	(*Valve 12, A+B*)
	(*spare*)
		Valve12FB
			(
			Enable_Motion:= Enable_Motion ,
			Enable_Latch:= TRUE,					(*Enabling Runs Valve as detent type (maintained solenoids*)
			Enable_SideA_PreCharge:= FALSE,		(*Enabling Turns Side A PreCharge Active, reset when Side B is energized in Auto*)
			Enable_SideB_PreCharge:= FALSE,		(*Enabling Turns Side B PreCharge Active, reset when Side A is energized in Auto*)
			PreCharge_Time:= T#0.10S,
			Enable_Auto_Commands:= Enable_Motion,
			Enable_Manual_Commands:= FALSE,
			In_Manual_SideA_Command:= FALSE,
			In_Manual_SideB_Command:= FALSE,
			SideA_Indicator:= FALSE,
			SideB_Indicator:= FALSE,
			TurnOn_SideA_SOL=> N100.Q.22,
			TurnOn_SideB_SOL=> N100.Q.23,
			TurnOn_SideA_Indicator=> ,
			TurnOn_SideB_Indicator=>
			 );
		Valve12FB.In_Auto_SideA_Command:= FALSE;
		Valve12FB.In_Auto_SideB_Command:= FALSE;


	(*Valve 13, A+B*)
	(*spare*)
		Valve13FB
			(
			Enable_Motion:= Enable_Motion ,
			Enable_Latch:= TRUE,					(*Enabling Runs Valve as detent type (maintained solenoids*)
			Enable_SideA_PreCharge:= FALSE,		(*Enabling Turns Side A PreCharge Active, reset when Side B is energized in Auto*)
			Enable_SideB_PreCharge:= FALSE,		(*Enabling Turns Side B PreCharge Active, reset when Side A is energized in Auto*)
			PreCharge_Time:= T#0.10S,
			Enable_Auto_Commands:= Enable_Motion,
			Enable_Manual_Commands:= FALSE,
			In_Manual_SideA_Command:= FALSE,
			In_Manual_SideB_Command:= FALSE,
			SideA_Indicator:= FALSE,
			SideB_Indicator:= FALSE,
			TurnOn_SideA_SOL=> N100.Q.24,
			TurnOn_SideB_SOL=> N100.Q.25,
			TurnOn_SideA_Indicator=> ,
			TurnOn_SideB_Indicator=>
			 );
		Valve13FB.In_Auto_SideA_Command:= FALSE;
		Valve13FB.In_Auto_SideB_Command:= FALSE;


	(*Valve 14, A+B*)
	(*spare*)
		Valve14FB
			(
			Enable_Motion:= Enable_Motion ,
			Enable_Latch:= TRUE,					(*Enabling Runs Valve as detent type (maintained solenoids*)
			Enable_SideA_PreCharge:= FALSE,		(*Enabling Turns Side A PreCharge Active, reset when Side B is energized in Auto*)
			Enable_SideB_PreCharge:= FALSE,		(*Enabling Turns Side B PreCharge Active, reset when Side A is energized in Auto*)
			PreCharge_Time:= T#0.10S,
			Enable_Auto_Commands:= Enable_Motion,
			Enable_Manual_Commands:= FALSE,
			In_Manual_SideA_Command:= FALSE,
			In_Manual_SideB_Command:= FALSE,
			SideA_Indicator:= FALSE,
			SideB_Indicator:= FALSE,
			TurnOn_SideA_SOL=> N100.Q.26,
			TurnOn_SideB_SOL=> N100.Q.27,
			TurnOn_SideA_Indicator=> ,
			TurnOn_SideB_Indicator=>
			 );
		Valve14FB.In_Auto_SideA_Command:= FALSE;
		Valve14FB.In_Auto_SideB_Command:= FALSE;


	(*Valve 15, A+B*)
	(*spare*)
		Valve15FB
			(
			Enable_Motion:= Enable_Motion ,
			Enable_Latch:= TRUE,					(*Enabling Runs Valve as detent type (maintained solenoids*)
			Enable_SideA_PreCharge:= FALSE,		(*Enabling Turns Side A PreCharge Active, reset when Side B is energized in Auto*)
			Enable_SideB_PreCharge:= FALSE,		(*Enabling Turns Side B PreCharge Active, reset when Side A is energized in Auto*)
			PreCharge_Time:= T#0.10S,
			Enable_Auto_Commands:= Enable_Motion,
			Enable_Manual_Commands:= FALSE,
			In_Manual_SideA_Command:= FALSE,
			In_Manual_SideB_Command:= FALSE,
			SideA_Indicator:= FALSE,
			SideB_Indicator:= FALSE,
			TurnOn_SideA_SOL=> N100.Q.28,
			TurnOn_SideB_SOL=> N100.Q.29,
			TurnOn_SideA_Indicator=> ,
			TurnOn_SideB_Indicator=>
			 );
		Valve15FB.In_Auto_SideA_Command:= FALSE;
		Valve15FB.In_Auto_SideB_Command:= FALSE;


	(*Valve 16, A+B*)
	(*spare*)
		Valve16FB
			(
			Enable_Motion:= Enable_Motion ,
			Enable_Latch:= TRUE,					(*Enabling Runs Valve as detent type (maintained solenoids*)
			Enable_SideA_PreCharge:= FALSE,		(*Enabling Turns Side A PreCharge Active, reset when Side B is energized in Auto*)
			Enable_SideB_PreCharge:= FALSE,		(*Enabling Turns Side B PreCharge Active, reset when Side A is energized in Auto*)
			PreCharge_Time:= T#0.10S,
			Enable_Auto_Commands:= Enable_Motion,
			Enable_Manual_Commands:= FALSE,
			In_Manual_SideA_Command:= FALSE,
			In_Manual_SideB_Command:= FALSE,
			SideA_Indicator:= FALSE,
			SideB_Indicator:= FALSE,
			TurnOn_SideA_SOL=> N100.Q.30,
			TurnOn_SideB_SOL=> N100.Q.31,
			TurnOn_SideA_Indicator=> ,
			TurnOn_SideB_Indicator=>
			 );
		Valve16FB.In_Auto_SideA_Command:= FALSE;
		Valve16FB.In_Auto_SideB_Command:= FALSE;


























(*end*)
END_ACTION

ACTION Xfer_To_UI:
	(*Transfer General Status and I/O Images for Display On HMI*)
	Discrete_Image.CLFaults1:= CLFaults1;
	Discrete_Image.CLFaults2:= CLFaults2;
	Discrete_Image.CLFaults3:= CLFaults3;
	Discrete_Image.CLFaults4:= CLFaults4;
	Discrete_Image.CLFaulted:= CLFaulted;
	Discrete_Image.PPFaults:= PPFaults;
	Discrete_Image.PPFaulted:= PPFaulted;

	Discrete_Image.N01:=N01;
	Discrete_Image.N02:=N02;
	Discrete_Image.N03:=N03;
	Discrete_Image.N04:=N04;
	Discrete_Image.N05:=N05;
	Discrete_Image.N06:=N06;
	Discrete_Image.N07:=N07;
	Discrete_Image.N08:=N08;
	Discrete_Image.N09:=N09;
	Discrete_Image.N100:=N100;
	Discrete_Image.N100_STAT:=N100_STAT;
	Discrete_Image.NodeLayout:=NodeLayout;
	Discrete_Image.NodeState:=NodeState;

	Discrete_Image.ID:= ID;
	Discrete_Image.ECatSlave_Cable_Breaks:= ECatSlave_Cable_Breaks;
	Discrete_Image.Input_Node_Count:= Input_Node_Count;
	Discrete_Image.VB_Node_Count:= VB_Node_Count;
















(*end*)
END_ACTION

END_PROGRAM

// ---- POUs/Fixtures and EOAT/Not_Used/EOAT10.TcPOU
(*EOAT*)


PROGRAM EOAT10

VAR_INPUT
(*General Inputs*)
	Enable_FB: BOOL;
	Enable_Motion: BOOL;
	Dry_Cycle: BOOL;
	NodeLayout:udt_ECATNodeData_20221507;
	ID: UINT;

	Input_Node_Count: UDINT;
	Output_Node_Count: UDINT;
	VB_Node_Count: UDINT;
	Robot_WorkingOK: BOOL;

(*CMDs (commands)*)
	CMD_CheckAllSensors_OFF: BOOL;
	CMD_CheckSensorsOFF_Grp1: BOOL;
	CMD_CheckSensorsOFF_Grp2: BOOL;
	CMD_CheckSensorsOFF_Grp3: BOOL;
	CMD_CheckSensorsOFF_Grp4: BOOL;
	CMD_CheckSensorsOFF_Grp5: BOOL;

	CMD_CheckAllSensors_ON: BOOL;
	CMD_CheckSensorsON_Grp1: BOOL;
	CMD_CheckSensorsON_Grp2: BOOL;
	CMD_CheckSensorsON_Grp3: BOOL;
	CMD_CheckSensorsON_Grp4: BOOL;
	CMD_CheckSensorsON_Grp5: BOOL;

	CMD_Tool_To_WORK: BOOL;
	CMD_CylToWORK_Grp1: BOOL;
	CMD_CylToWORK_Grp2: BOOL;
	CMD_CylToWORK_Grp3: BOOL;
	CMD_CylToWORK_Grp4: BOOL;
	CMD_CylToWORK_Grp5: BOOL;

	CMD_Tool_To_HOME: BOOL;
	CMD_CylToHOME_Grp1: BOOL;
	CMD_CylToHOME_Grp2: BOOL;
	CMD_CylToHOME_Grp3: BOOL;
	CMD_CylToHOME_Grp4: BOOL;
	CMD_CylToHOME_Grp5: BOOL;


END_VAR

VAR
(*Hardware Related Data Types*)
			(*Develop "Beckhoff Nodes"*)
			{attribute 'OPC.UA.DA':='1'}
			N01 AT %I*: udt_EP1008_002_v2;
			{attribute 'OPC.UA.DA':='1'}
			N02 AT %I*: udt_EP1008_002_v2;
			{attribute 'OPC.UA.DA':='1'}
			N03 AT %I*: udt_EP1008_002_v2;
			{attribute 'OPC.UA.DA':='1'}
			N04 AT %I*: udt_EP1008_002_v2;
			{attribute 'OPC.UA.DA':='1'}
			N05 AT %I*: udt_EP1008_002_v2;
			{attribute 'OPC.UA.DA':='1'}
			N06 AT %I*: udt_EP1008_002_v2;
			{attribute 'OPC.UA.DA':='1'}
			N07 AT %I*: udt_EP1008_002_v2;
			{attribute 'OPC.UA.DA':='1'}
			N08 AT %I*: udt_EP1008_002_v2;
			{attribute 'OPC.UA.DA':='1'}
			N09 AT %I*: udt_EP1008_002_v2;
			{attribute 'OPC.UA.DA':='1'}
			N100 AT %Q*: udt_SMC_EX260_ValveBank;
			{attribute 'OPC.UA.DA':='1'}
			N100_STAT AT %I*:udt_SMC_EX260_Stat;

(* Nodes States*)
	NodeState: ARRAY[0..63] OF UINT;
	DiscreteNode_OK: BOOL;
(* Cable Break States*)
	ECatSlave_Cable_Breaks: ARRAY[0..1]OF DINT;

(*Standard Internal Variables*)
		(*Generic Sensor Variables*)
		All_Sensors_On: UINT;
		All_Sensors_Off: UINT;
		(*Generic Position Variables*)
		Tool_At_Home: UINT;
		Tool_At_Work: UINT;
		(*General Internals*)
		CLFaulted: UDINT;
		PPFaulted: UDINT;

(*Non-Standard Variables*)

		(*FB Instances*)
		Clamp1FB: FB_Cylinder_Status;
		Clamp2FB: FB_Cylinder_Status;
		Clamp3FB: FB_Cylinder_Status;
		Clamp4FB: FB_Cylinder_Status;
		Clamp5FB: FB_Cylinder_Status;
		Clamp6FB: FB_Cylinder_Status;
		Clamp7FB: FB_Cylinder_Status;
		Clamp8FB: FB_Cylinder_Status;
		Clamp9FB: FB_Cylinder_Status;
		Clamp10FB: FB_Cylinder_Status;
		Clamp11FB: FB_Cylinder_Status;
		Clamp12FB: FB_Cylinder_Status;
		Pin1FB: FB_Cylinder_Status;
		Pin2FB: FB_Cylinder_Status;
		Pin3FB: FB_Cylinder_Status;
		Pin4FB: FB_Cylinder_Status;
		Pin5FB: FB_Cylinder_Status;
		Pin6FB: FB_Cylinder_Status;

		Part_Present1FB: FB_PP_Sensor;
		Part_Present2FB: FB_PP_Sensor;
		Part_Present3FB: FB_PP_Sensor;
		Part_Present4FB: FB_PP_Sensor;
		Part_Present5FB: FB_PP_Sensor;
		Part_Present6FB: FB_PP_Sensor;
		Part_Present7FB: FB_PP_Sensor;
		Part_Present8FB: FB_PP_Sensor;

		(*Valve FBs*)
		Valve1FB: FB_GTAC_Valve_20170704;
		Valve2FB: FB_GTAC_Valve_20170704;
		Valve3FB: FB_GTAC_Valve_20170704;
		Valve4FB: FB_GTAC_Valve_20170704;
		Valve5FB: FB_GTAC_Valve_20170704;
		Valve6FB: FB_GTAC_Valve_20170704;
		Valve7FB: FB_GTAC_Valve_20170704;
		Valve8FB: FB_GTAC_Valve_20170704;
		Valve9FB: FB_GTAC_Valve_20170704;
		Valve10FB: FB_GTAC_Valve_20170704;
		Valve11FB: FB_GTAC_Valve_20170704;
		Valve12FB: FB_GTAC_Valve_20170704;
		Valve13FB: FB_GTAC_Valve_20170704;
		Valve14FB: FB_GTAC_Valve_20170704;
		Valve15FB: FB_GTAC_Valve_20170704;
		Valve16FB: FB_GTAC_Valve_20170704;

		(*Tool Positions*)
		Clamp1ADVD: BOOL;
		Clamp1RETD: BOOL;
		Clamp2ADVD: BOOL;
		Clamp2RETD: BOOL;
		Clamp3ADVD: BOOL;
		Clamp3RETD: BOOL;
		Clamp4ADVD: BOOL;
		Clamp4RETD: BOOL;
		Clamp5ADVD: BOOL;
		Clamp5RETD: BOOL;
		Clamp6ADVD: BOOL;
		Clamp6RETD: BOOL;
		Clamp7ADVD: BOOL;
		Clamp7RETD: BOOL;
		Clamp8ADVD: BOOL;
		Clamp8RETD: BOOL;
		Clamp9ADVD: BOOL;
		Clamp9RETD: BOOL;
		Clamp10ADVD: BOOL;
		Clamp10RETD: BOOL;
		Clamp11ADVD: BOOL;
		Clamp11RETD: BOOL;
		Clamp12ADVD: BOOL;
		Clamp12RETD: BOOL;
		Pin1ADVD: BOOL;
		Pin1RETD: BOOL;
		Pin2ADVD: BOOL;
		Pin2RETD: BOOL;
		Pin3ADVD: BOOL;
		Pin3RETD: BOOL;
		Pin4ADVD: BOOL;
		Pin4RETD: BOOL;
		Pin5ADVD: BOOL;
		Pin5RETD: BOOL;
		Pin6ADVD: BOOL;
		Pin6RETD: BOOL;

		(*Part Present Sensors*)
		(*Main Body Present*)
		Part_Present1: BOOL;
		Part_Present2: BOOL;
		Part_Present3: BOOL;
		Part_Present4: BOOL;
		Part_Present5: BOOL;
		Part_Present6: BOOL;
		Part_Present7: BOOL;
		Part_Present8: BOOL;



END_VAR

VAR_OUTPUT

		FB_OK: BOOL;
		Discrete_Image: udt_EOATxx_Image_20170607;

		EOAT_FLT: BOOL;

		CLFaults1:UDINT;
		CLFaults2:UDINT;
		CLFaults3:UDINT;
		CLFaults4:UDINT;
		PPFaults: UDINT;

		EOAT_All_Empty: BOOL;
		EOAT_Part1_Empty: BOOL;
		EOAT_Part2_Empty: BOOL;
		EOAT_Part3_Empty: BOOL;
		EOAT_Part4_Empty: BOOL;
		EOAT_Part5_Empty: BOOL;

		EOAT_Full: BOOL;
		Part1_In_EOAT: BOOL;
		Part2_In_EOAT: BOOL;
		Part3_In_EOAT: BOOL;
		Part4_In_EOAT: BOOL;
		Part5_In_EOAT: BOOL;

	(*ACKS*)
		ACK_Tool_At_WORK: BOOL;
		ACK_CylAtWORK_Grp1: BOOL;
		ACK_CylAtWORK_Grp2: BOOL;
		ACK_CylAtWORK_Grp3: BOOL;
		ACK_CylAtWORK_Grp4: BOOL;
		ACK_CylAtWORK_Grp5: BOOL;
	
		ACK_Tool_At_HOME: BOOL;
		ACK_CylAtHOME_Grp1: BOOL;
		ACK_CylAtHOME_Grp2: BOOL;
		ACK_CylAtHOME_Grp3: BOOL;
		ACK_CylAtHOME_Grp4: BOOL;
		ACK_CylAtHOME_Grp5: BOOL;


END_VAR

	(*Set FB_OK to True*)
	FB_OK:= TRUE;


(*---------------------------------------------------- Gather Hardwear ------------------------------------------------------*)
	Hardware();


(*---------------------------------------------------- Gather Clamp Sensor Inputs --------------------------------------*)
	Cylinders();


(*---------------------------------------------------- Gather Part Present Sensor Inputs ------------------------------*)
	Proxies();


(*---------------------------------------------------- Group Clamp Sensors -----------------------------------------------*)
	Tool_States();


(*---------------------------------------------------- Group Part Present Sensors ---------------------------------------*)
	All_Sensors();



(*---------------------------------------------------- Status and Faults--------------------------------------------------------*)
	Status_and_Faults();


(*---------------------------------------------------- Transfer to UI -------------------------------------------------------------*)
	Xfer_To_UI();


(*------------------------------------------------------Transfer Valve Outputs ----------------------------------------------*)
	ValveBank1();


(*---------------------------------------------------- Gather Robot Registration-------------------------------------------*)









(*end*)

ACTION All_Sensors:


(*	Note - In the event there is a left part and a right part, grouping the sensors allows only portions of the sensors to be monitored at a time.
		If this is not advantageous to the design, there is still the option to group all the sensors as one group instead.
		In this example, there are all 5 groups set up. 
		Change this section to suit the specific design you have, where .0 is all, .1 is group one, .2 is group two, etc*)


	(*All Sensors Off*)
	All_Sensors_Off.0:= NOT Part_Present1 AND NOT Part_Present2 AND NOT  Part_Present3
					AND NOT Part_Present4 AND NOT Part_Present5 AND NOT Part_Present6
					AND NOT Part_Present7 AND NOT Part_Present8;

	(*All Sensors Off - Group 1*)
	All_Sensors_Off.1:= NOT Part_Present1 AND NOT Part_Present2 AND NOT  Part_Present3
					AND NOT Part_Present4 AND NOT Part_Present5;

	(*All Sensors Off - Group 2*)
	All_Sensors_Off.2:= NOT Part_Present6 AND NOT Part_Present7 AND NOT Part_Present8;

	(*All Sensors Off - Group 3*)
	All_Sensors_Off.3:= FALSE;

	(*All Sensors Off - Group 4*)
	All_Sensors_Off.4:= FALSE;

	(*All Sensors Off - Group 5*)
	All_Sensors_Off.5:= FALSE;



	(*All Sensors On*)
	All_Sensors_On.0:= (Part_Present1 AND Part_Present2 AND Part_Present3
					AND Part_Present4 AND Part_Present5 AND Part_Present6
					AND Part_Present7 AND Part_Present8)
					OR (All_Sensors_Off.0 AND Dry_Cycle);

	(*All Sensors On - Group 1*)
	All_Sensors_On.1:= (Part_Present1 AND Part_Present2 AND Part_Present3 AND Part_Present4 AND Part_Present5)
					OR (All_Sensors_Off.0 AND Dry_Cycle);

	(*All Sensors On - Group 2*)
	All_Sensors_On.2:= (Part_Present6 AND Part_Present7 AND Part_Present8)
					OR (All_Sensors_Off.0 AND Dry_Cycle);

	(*All Sensors On - Group 3*)
	All_Sensors_On.3:= (FALSE)
					OR (All_Sensors_Off.0 AND Dry_Cycle);

	(*All Sensors On - Group 4*)
	All_Sensors_On.4:= (FALSE)
					OR (All_Sensors_Off.0 AND Dry_Cycle);

	(*All Sensors On - Group 5*)
	All_Sensors_On.5:= (FALSE)
					OR (All_Sensors_Off.0 AND Dry_Cycle);




	(*Group all Sensors*)
	IF CMD_CheckAllSensors_OFF AND All_Sensors_Off.0
		THEN
			EOAT_All_Empty:= TRUE;
			EOAT_Full:= FALSE;

	ELSIF CMD_CheckAllSensors_ON AND All_Sensors_On.0
		THEN
			EOAT_All_Empty:= FALSE;
			EOAT_Full:= TRUE;

	END_IF

	IF CMD_CheckSensorsOFF_Grp1 AND All_Sensors_Off.1
		THEN
			EOAT_Part1_Empty:= TRUE;
			Part1_In_EOAT:= FALSE;

	ELSIF CMD_CheckSensorsON_Grp1 AND All_Sensors_On.1
		THEN
			EOAT_Part1_Empty:= FALSE;
			Part1_In_EOAT:= TRUE;

	END_IF

	IF CMD_CheckSensorsOFF_Grp2 AND All_Sensors_Off.2
		THEN
			EOAT_Part2_Empty:= TRUE;
			Part2_In_EOAT:= FALSE;

	ELSIF CMD_CheckSensorsON_Grp2 AND All_Sensors_On.2
		THEN
			EOAT_Part2_Empty:= FALSE;
			Part2_In_EOAT:= TRUE;

	END_IF

	IF CMD_CheckSensorsOFF_Grp3 AND All_Sensors_Off.3
		THEN
			EOAT_Part3_Empty:= TRUE;
			Part3_In_EOAT:= FALSE;

	ELSIF CMD_CheckSensorsON_Grp3 AND All_Sensors_On.3
		THEN
			EOAT_Part3_Empty:= FALSE;
			Part3_In_EOAT:= TRUE;

	ELSIF CMD_CheckSensorsON_Grp3 AND All_Sensors_On.3
		THEN
			EOAT_Part3_Empty:= FALSE;
			Part3_In_EOAT:= TRUE;

	END_IF

	IF CMD_CheckSensorsOFF_Grp4 AND All_Sensors_Off.4
		THEN
			EOAT_Part4_Empty:= TRUE;
			Part4_In_EOAT:= FALSE;
	ELSIF CMD_CheckSensorsON_Grp4 AND All_Sensors_On.4
		THEN
			EOAT_Part4_Empty:= FALSE;
			Part4_In_EOAT:= TRUE;

	END_IF

	IF CMD_CheckSensorsOFF_Grp5 AND All_Sensors_Off.5
		THEN
			EOAT_Part5_Empty:= TRUE;
			Part5_In_EOAT:= FALSE;
	ELSIF CMD_CheckSensorsON_Grp5 AND All_Sensors_On.5
		THEN
			EOAT_Part5_Empty:= FALSE;
			Part5_In_EOAT:= TRUE;

	END_IF












(*end*)
END_ACTION

ACTION Cylinders:
(*Clamps*)(*Clamps*)(*Clamps*)
(*Clamps*)(*Clamps*)(*Clamps*)
(*Clamps*)(*Clamps*)(*Clamps*)

		(*Clamp1*)
		Clamp1FB(
			Retracted_Sensor:= N02.I.0,
			Advanced_Sensor:= N02.I.1,
			Retract_Solenoid:= N100.Q.1,
			Advance_Solenoid:= N100.Q.0,
			Ret_Delay:= T#0.1s,
			Adv_Delay:= T#0.1s,
			Fault_Delay:= T#3s,
			Disable_Fault:= FALSE,
			In_Retracted_Position=> Clamp1RETD,
			In_Advanced_Position=> Clamp1ADVD,
			Faulted=> CLFaults1.1 );

		(*Clamp2 *)
		Clamp2FB(
			Retracted_Sensor:= N02.I.2,
			Advanced_Sensor:= N02.I.3,
			Retract_Solenoid:= N100.Q.1,
			Advance_Solenoid:= N100.Q.0,
			Ret_Delay:= T#0.1s,
			Adv_Delay:= T#0.1s,
			Fault_Delay:= T#3s,
			Disable_Fault:= FALSE,
			In_Retracted_Position=> Clamp2RETD,
			In_Advanced_Position=> Clamp2ADVD,
			Faulted=> CLFaults1.2 );

		(*Clamp3 *)
		Clamp3FB(
			Retracted_Sensor:= N02.I.4,
			Advanced_Sensor:= N02.I.5,
			Retract_Solenoid:= N100.Q.5,
			Advance_Solenoid:= N100.Q.4,
			Ret_Delay:= T#0.1s,
			Adv_Delay:= T#0.1s,
			Fault_Delay:= T#3s,
			Disable_Fault:= FALSE,
			In_Retracted_Position=> Clamp3RETD,
			In_Advanced_Position=> Clamp3ADVD,
			Faulted=> CLFaults1.3 );

		(*Clamp4 *)
		Clamp4FB(
			Retracted_Sensor:= N02.I.6,
			Advanced_Sensor:= N02.I.7,
			Retract_Solenoid:= N100.Q.1,
			Advance_Solenoid:= N100.Q.0,
			Ret_Delay:= T#0.1s,
			Adv_Delay:= T#0.1s,
			Fault_Delay:= T#3s,
			Disable_Fault:= FALSE,
			In_Retracted_Position=> Clamp4RETD,
			In_Advanced_Position=> Clamp4ADVD,
			Faulted=> CLFaults1.4 );

		(*Clamp5 *)
		Clamp5FB(
			Retracted_Sensor:= N03.I.0,
			Advanced_Sensor:= N03.I.1,
			Retract_Solenoid:= N100.Q.15,
			Advance_Solenoid:= N100.Q.14,
			Ret_Delay:= T#0.1s,
			Adv_Delay:= T#0.1s,
			Fault_Delay:= T#3s,
			Disable_Fault:= FALSE,
			In_Retracted_Position=> Clamp5RETD,
			In_Advanced_Position=> Clamp5ADVD,
			Faulted=> CLFaults2.5 );

		(*Clamp6 *)
		Clamp6FB(
			Retracted_Sensor:= N03.I.2,
			Advanced_Sensor:= N03.I.3,
			Retract_Solenoid:= N100.Q.11,
			Advance_Solenoid:= N100.Q.10,
			Ret_Delay:= T#0.1s,
			Adv_Delay:= T#0.1s,
			Fault_Delay:= T#3s,
			Disable_Fault:= FALSE,
			In_Retracted_Position=> Clamp6RETD,
			In_Advanced_Position=> Clamp6ADVD,
			Faulted=> CLFaults2.6 );

		(*Clamp7 *)
		Clamp7FB(
			Retracted_Sensor:= N03.I.4,
			Advanced_Sensor:= N03.I.5,
			Retract_Solenoid:= N100.Q.15,
			Advance_Solenoid:= N100.Q.14,
			Ret_Delay:= T#0.1s,
			Adv_Delay:= T#0.1s,
			Fault_Delay:= T#3s,
			Disable_Fault:= FALSE,
			In_Retracted_Position=> Clamp7RETD,
			In_Advanced_Position=> Clamp7ADVD,
			Faulted=> CLFaults2.7 );

		(*Clamp8 *)
		Clamp8FB(
			Retracted_Sensor:= N03.I.6,
			Advanced_Sensor:= N03.I.7,
			Retract_Solenoid:= N100.Q.15,
			Advance_Solenoid:= N100.Q.14,
			Ret_Delay:= T#0.1s,
			Adv_Delay:= T#0.1s,
			Fault_Delay:= T#3s,
			Disable_Fault:= FALSE,
			In_Retracted_Position=> Clamp8RETD,
			In_Advanced_Position=> Clamp8ADVD,
			Faulted=> CLFaults2.8 );

		(*Clamp9*)
		Clamp9FB(
			Retracted_Sensor:= N04.I.0,
			Advanced_Sensor:= N04.I.1,
			Retract_Solenoid:= N100.Q.1,
			Advance_Solenoid:= N100.Q.0,
			Ret_Delay:= T#0.1s,
			Adv_Delay:= T#0.1s,
			Fault_Delay:= T#3s,
			Disable_Fault:= FALSE,
			In_Retracted_Position=> Clamp9RETD,
			In_Advanced_Position=> Clamp9ADVD,
			Faulted=> CLFaults2.9 );

		(*Clamp10*)
		Clamp10FB(
			Retracted_Sensor:= N04.I.2,
			Advanced_Sensor:= N04.I.3,
			Retract_Solenoid:= N100.Q.1,
			Advance_Solenoid:= N100.Q.0,
			Ret_Delay:= T#0.1s,
			Adv_Delay:= T#0.1s,
			Fault_Delay:= T#3s,
			Disable_Fault:= FALSE,
			In_Retracted_Position=> Clamp10RETD,
			In_Advanced_Position=> Clamp10ADVD,
			Faulted=> CLFaults2.10 );

		(*Clamp11*)
		Clamp11FB(
			Retracted_Sensor:= N04.I.4,
			Advanced_Sensor:= N04.I.5,
			Retract_Solenoid:= N100.Q.1,
			Advance_Solenoid:= N100.Q.0,
			Ret_Delay:= T#0.1s,
			Adv_Delay:= T#0.1s,
			Fault_Delay:= T#3s,
			Disable_Fault:= FALSE,
			In_Retracted_Position=> Clamp11RETD,
			In_Advanced_Position=> Clamp11ADVD,
			Faulted=> CLFaults2.11 );

		(*Clamp12*)
		Clamp12FB(
			Retracted_Sensor:= N04.I.6,
			Advanced_Sensor:= N04.I.7,
			Retract_Solenoid:= N100.Q.1,
			Advance_Solenoid:= N100.Q.0,
			Ret_Delay:= T#0.1s,
			Adv_Delay:= T#0.1s,
			Fault_Delay:= T#3s,
			Disable_Fault:= FALSE,
			In_Retracted_Position=> Clamp12RETD,
			In_Advanced_Position=> Clamp12ADVD,
			Faulted=> CLFaults2.12 );


(*Pins*)(*Pins*)(*Pins*)
(*Pins*)(*Pins*)(*Pins*)
(*Pins*)(*Pins*)(*Pins*)

		(*Pin1*)
		Pin1FB(
			Retracted_Sensor:=  N03.I.0,
			Advanced_Sensor:=  N03.I.1,
			Retract_Solenoid:=  N100.Q.7,
			Advance_Solenoid:=  N100.Q.6,
			Adv_Delay:=  T#0.1S,
			Ret_Delay:=  T#0.1S,
			Fault_Delay:=  T#3.0S,
			Disable_Fault:= FALSE,
			In_Retracted_Position=> Pin1RETD,
			In_Advanced_Position=> Pin1ADVD,
			Faulted=> CLFaults1.5);

		(*Pin2*)
		Pin2FB(
			Retracted_Sensor:=  N03.I.2,
			Advanced_Sensor:=  N03.I.3,
			Retract_Solenoid:=  N100.Q.7,
			Advance_Solenoid:=  N100.Q.6,
			Adv_Delay:=  T#0.1S,
			Ret_Delay:=  T#0.1S,
			Fault_Delay:=  T#3.0S,
			Disable_Fault:= FALSE,
			In_Retracted_Position=> Pin2RETD,
			In_Advanced_Position=> Pin2ADVD,
			Faulted=> CLFaults1.6);

		(*Pin3*)
		Pin3FB(
			Retracted_Sensor:=  N03.I.4,
			Advanced_Sensor:=  N03.I.5,
			Retract_Solenoid:=  N100.Q.7,
			Advance_Solenoid:=  N100.Q.6,
			Adv_Delay:=  T#0.1S,
			Ret_Delay:=  T#0.1S,
			Fault_Delay:=  T#3.0S,
			Disable_Fault:= FALSE,
			In_Retracted_Position=> Pin3RETD,
			In_Advanced_Position=> Pin3ADVD,
			Faulted=> CLFaults1.7 );

		(*Pin4*)
		Pin4FB(
			Retracted_Sensor:=  N03.I.6,
			Advanced_Sensor:=  N03.I.7,
			Retract_Solenoid:=  N100.Q.13,
			Advance_Solenoid:=  N100.Q.12,
			Adv_Delay:=  T#0.1S,
			Ret_Delay:=  T#0.1S,
			Fault_Delay:=  T#3.0S,
			Disable_Fault:= FALSE,
			In_Retracted_Position=> Pin4RETD,
			In_Advanced_Position=> Pin4ADVD,
			Faulted=> CLFaults1.8 );

		(*Pin5*)
		Pin5FB(
			Retracted_Sensor:=  N04.I.0,
			Advanced_Sensor:=  N04.I.1,
			Retract_Solenoid:=  N100.Q.13,
			Advance_Solenoid:=  N100.Q.12,
			Adv_Delay:=  T#0.1S,
			Ret_Delay:=  T#0.1S,
			Fault_Delay:=  T#3.0S,
			Disable_Fault:= FALSE,
			In_Retracted_Position=> Pin5RETD,
			In_Advanced_Position=> Pin5ADVD,
			Faulted=> CLFaults1.9);

		(*Pin6*)
		Pin6FB(
			Retracted_Sensor:=  N04.I.2,
			Advanced_Sensor:=  N04.I.3,
			Retract_Solenoid:=  N100.Q.13,
			Advance_Solenoid:=  N100.Q.12,
			Adv_Delay:=  T#0.1S,
			Ret_Delay:=  T#0.1S,
			Fault_Delay:=  T#3.0S,
			Disable_Fault:= FALSE,
			In_Retracted_Position=> Pin6RETD,
			In_Advanced_Position=> Pin6ADVD,
			Faulted=> CLFaults1.10 );

































(*end*)
END_ACTION

ACTION Hardware:
(*Pass Node States into Array  in order on Physical Fixture*)

	NodeState:=NodeLayout.State;

(*$$$$$$$$$$$$$$$$$$$$$$$$$$$$$$$$$$$$$$$$$$$$$$$$Gather Status Of Hardware $$$$$$$$$$$$$$$$$$$$$$$$$$$$$$$$$$$$$$$$$$$$$$$$$$$$*)
	(*Discrete I/O Nodes*)

	IF (N01.InfoData.State=8)
		AND (N01.InfoData.State=8 OR (Input_Node_Count<2))
		AND (N02.InfoData.State=8 OR (Input_Node_Count<3))
		AND (N03.InfoData.State=8 OR (Input_Node_Count<4))
		AND (N04.InfoData.State=8 OR (Input_Node_Count<5))
		AND (N05.InfoData.State=8 OR (Input_Node_Count<6))
		AND (N06.InfoData.State=8 OR (Input_Node_Count<7))
		AND (N07.InfoData.State=8 OR (Input_Node_Count<8))
		AND (N08.InfoData.State=8 OR (Input_Node_Count<9))
		AND (N09.InfoData.State=8 OR (Input_Node_Count<10))
		AND (N100_STAT.InfoData.State=8)

		THEN
			DiscreteNode_OK:=TRUE;

	ELSE
			DiscreteNode_OK:=FALSE;

	END_IF;

	(*Cable Break Detection*)
		ECatSlave_Cable_Breaks:= FUN_GTAC_EcatSlaveConnState_64bit(NodeState);		(*Function Returns Flags to warn of possible cable break*)
END_ACTION

ACTION Proxies:


(*+++++++++++THIS AREA IS CUSTOM PER INSTALLATION AND WILL HAVE TO BE MODIFIED PER +++++++++++++*)
(*+++++++++++THIS AREA IS CUSTOM PER INSTALLATION AND WILL HAVE TO BE MODIFIED PER +++++++++++++*)

(*Note - On_Trigger and Off_Trigger need to be changed based on which group in All_Sensors_On the sensor is placed.*)


	(*Part 1 Present*)
		Part_Present1FB(
			Sensor_Input:= N01.I.0,
			On_Trigger1:= CMD_CheckAllSensors_ON OR CMD_CheckSensorsON_Grp1 OR EOAT_Full OR Part1_In_EOAT,
			On_Trigger2:= TRUE,
			Off_Trigger1:= CMD_CheckAllSensors_OFF OR CMD_CheckSensorsOFF_Grp1 OR EOAT_All_Empty OR EOAT_Part1_Empty,
			Off_Trigger2:= TRUE,
			Disable_Faults:= Dry_Cycle OR Robot_WorkingOK,
			Fault_Delay:= T#1.5s,
			Status=> Part_Present1,
			Faulted=>  PPFaults.1);

	(*Part 2 Present*)
		Part_Present2FB(
			Sensor_Input:= N01.I.1,
			On_Trigger1:= CMD_CheckAllSensors_ON OR CMD_CheckSensorsON_Grp1,
			On_Trigger2:= TRUE,
			Off_Trigger1:= CMD_CheckAllSensors_OFF OR CMD_CheckSensorsOFF_Grp1,
			Off_Trigger2:= TRUE,
			Disable_Faults:= Dry_Cycle OR Robot_WorkingOK,
			Fault_Delay:= T#1.5s,
			Status=> Part_Present2,
			Faulted=>  PPFaults.2);

	(*Part 3 Present*)
		Part_Present3FB(
			Sensor_Input:= N01.I.2,
			On_Trigger1:= CMD_CheckAllSensors_ON OR CMD_CheckSensorsON_Grp1,
			On_Trigger2:= TRUE,
			Off_Trigger1:= CMD_CheckAllSensors_OFF OR CMD_CheckSensorsOFF_Grp1,
			Off_Trigger2:= TRUE,
			Disable_Faults:= Dry_Cycle OR Robot_WorkingOK,
			Fault_Delay:= T#1.5s,
			Status=> Part_Present3,
			Faulted=>  PPFaults.3);

	(*Part 4 Present*)
		Part_Present4FB(
			Sensor_Input:=N01.I.3,
			On_Trigger1:= CMD_CheckAllSensors_ON OR CMD_CheckSensorsON_Grp1,
			On_Trigger2:= TRUE,
			Off_Trigger1:= CMD_CheckAllSensors_OFF OR CMD_CheckSensorsOFF_Grp1,
			Off_Trigger2:= TRUE,
			Disable_Faults:= Dry_Cycle OR Robot_WorkingOK,
			Fault_Delay:= T#1.5s,
			Status=> Part_Present4,
			Faulted=>  PPFaults.4);

	(*Part 5 Present*)
		Part_Present5FB(
			Sensor_Input:= N01.I.4,
			On_Trigger1:= CMD_CheckAllSensors_ON OR CMD_CheckSensorsON_Grp1,
			On_Trigger2:= TRUE,
			Off_Trigger1:= CMD_CheckAllSensors_OFF OR CMD_CheckSensorsOFF_Grp1,
			Off_Trigger2:= TRUE,
			Disable_Faults:= Dry_Cycle OR Robot_WorkingOK,
			Fault_Delay:= T#1.5s,
			Status=> Part_Present5,
			Faulted=>  PPFaults.5);

	(*Part 6 Present*)
		Part_Present6FB(
			Sensor_Input:= N01.I.5,
			On_Trigger1:= CMD_CheckAllSensors_ON OR CMD_CheckSensorsON_Grp2,
			On_Trigger2:= TRUE,
			Off_Trigger1:= CMD_CheckAllSensors_OFF OR CMD_CheckSensorsOFF_Grp2,
			Off_Trigger2:= TRUE,
			Disable_Faults:= Dry_Cycle OR Robot_WorkingOK,
			Fault_Delay:= T#1.5s,
			Status=> Part_Present6,
			Faulted=>  PPFaults.6);

	(*Part 7 Present*)
		Part_Present7FB(
			Sensor_Input:= N01.I.7,
			On_Trigger1:= CMD_CheckAllSensors_ON OR CMD_CheckSensorsON_Grp2,
			On_Trigger2:= TRUE,
			Off_Trigger1:= CMD_CheckAllSensors_OFF OR CMD_CheckSensorsOFF_Grp2,
			Off_Trigger2:= TRUE,
			Disable_Faults:= Dry_Cycle OR Robot_WorkingOK,
			Fault_Delay:= T#1.5s,
			Status=> Part_Present7,
			Faulted=>  PPFaults.7);

	(*Part 8 Present*)
		Part_Present8FB(
			Sensor_Input:= N09.I.0,
			On_Trigger1:= CMD_CheckAllSensors_ON OR CMD_CheckSensorsON_Grp2,
			On_Trigger2:= TRUE,
			Off_Trigger1:= CMD_CheckAllSensors_OFF OR CMD_CheckSensorsOFF_Grp2,
			Off_Trigger2:= TRUE,
			Disable_Faults:= Dry_Cycle OR Robot_WorkingOK,
			Fault_Delay:= T#1.5s,
			Status=> Part_Present8,
			Faulted=>  PPFaults.8);


















(*end*)
END_ACTION

ACTION Status_and_Faults:
	(*Clamp/Cylinder Faults*)
		IF CLFaults1>0
			THEN CLFaulted.1:=TRUE;
		ELSE
			CLFaulted.1:=FALSE;
		END_IF;
	(*Spare Fault Word*)
		IF CLFaults2>0
			THEN CLFaulted.2:=TRUE;
		ELSE
			CLFaulted.2:=FALSE;
		END_IF;
	(*Spare Fault Word*)
		IF CLFaults3>0
			THEN CLFaulted.3:=TRUE;
		ELSE
			CLFaulted.3:=FALSE;
		END_IF;
	(*Spare Fault Word*)
		IF CLFaults4>0
			THEN CLFaulted.4:=TRUE;
		ELSE
			CLFaulted.4:=FALSE;
		END_IF;
	(*Bit 0 is designated as ANY Clamp Fault Word Faulted*)
		IF CLFaulted.1 OR CLFaulted.2 OR CLFaulted.3
			THEN CLFaulted.0:= TRUE;
		ELSE
			CLFaulted.0 := FALSE;
		END_IF;

	(*Part Present Sensor Faults*)
		IF PPFaults>0
			THEN PPFaulted.0:=TRUE;
		ELSE
			PPFaulted.0:=FALSE;
		END_IF;

		EOAT_FLT:= (CLFaulted>0) OR (PPFaulted>0);















(*end*)
END_ACTION

ACTION Tool_States:
(*	Note - In the event there is a left part and a right part, grouping the cylinders allows only portions of the cylinders to be controlled at a time.
		If this is not advantageous to the design, there is still the option to group all the cylinders as one group instead.
		In this example, there are all 5 groups set up. 
		Change this section to suit the specific design you have, where .0 is all, .1 is group one, .2 is group two, etc*)


	(*Tool All Home - All Cylinders Home*)
	Tool_At_Home.0:=Clamp1RETD AND Clamp2RETD AND Clamp3RETD AND Clamp4RETD
				AND Clamp5RETD AND Clamp6RETD AND Clamp7RETD AND Clamp8RETD
				AND Clamp9RETD AND Clamp10RETD AND Clamp11RETD AND Clamp12RETD
				AND Pin1ADVD AND Pin2ADVD AND Pin3ADVD AND Pin4ADVD AND Pin5ADVD AND Pin6ADVD;

	(*Tool All Home - Cylinders Home Group 1*)
	Tool_At_Home.1:=Clamp1RETD AND Clamp2RETD AND Clamp3RETD AND Clamp4RETD
				AND Clamp5RETD AND Clamp6RETD AND Clamp7RETD AND Clamp8RETD
				AND Clamp9RETD AND Clamp10RETD AND Clamp11RETD AND Clamp12RETD
				AND Pin1ADVD AND Pin2ADVD AND Pin3ADVD AND Pin4ADVD AND Pin5ADVD AND Pin6ADVD;

	(*Tool All Home - Cylinders Home Group 2*)
	Tool_At_Home.2:=Clamp1RETD AND Clamp2RETD AND Clamp3RETD AND Clamp4RETD
				AND Clamp5RETD AND Clamp6RETD AND Clamp7RETD AND Clamp8RETD
				AND Clamp9RETD AND Clamp10RETD AND Clamp11RETD AND Clamp12RETD
				AND Pin1ADVD AND Pin2ADVD AND Pin3ADVD AND Pin4ADVD AND Pin5ADVD AND Pin6ADVD;

	(*Tool All Home - Cylinders Home Group 3*)
	Tool_At_Home.3:= FALSE;

	(*Tool All Home - Cylinders Home Group 4*)
	Tool_At_Home.4:= FALSE;

	(*Tool All Home - Cylinders Home Group 5*)
	Tool_At_Home.5:= FALSE;




	(*Tool at Work - All Cylinders Work*)
	Tool_At_Work.0:= Clamp1ADVD AND Clamp2ADVD AND Clamp3ADVD AND Clamp4ADVD
				AND Clamp5ADVD AND Clamp6ADVD AND Clamp7ADVD AND Clamp8ADVD
				AND Clamp9ADVD AND Clamp10ADVD AND Clamp11ADVD AND Clamp12ADVD
				AND Pin1ADVD AND Pin2ADVD AND Pin3ADVD AND Pin4ADVD AND Pin5ADVD AND Pin6ADVD;

	(*Tool at Work - Cylinders Work Group 1*)
	Tool_At_Work.1:= Clamp1ADVD AND Clamp2ADVD AND Clamp3ADVD AND Clamp4ADVD
				AND Clamp5ADVD AND Clamp6ADVD AND Clamp7ADVD AND Clamp8ADVD;

	(*Tool at Work - Cylinders Work Group 2*)
	Tool_At_Work.2:= Clamp9ADVD AND Clamp10ADVD AND Clamp11ADVD AND Clamp12ADVD
				AND Pin1RETD AND Pin2RETD AND Pin3RETD AND Pin4RETD AND Pin5RETD AND Pin6RETD;

	(*Tool at Work - Cylinders Work Group 3*)
	Tool_At_Work.3:= FALSE;

	(*Tool at Work - Cylinders Work Group 4*)
	Tool_At_Work.4:= FALSE;

	(*Tool at Work - Cylinders Work Group 5*)
	Tool_At_Work.5:= FALSE;




	(*Group all Tool States*)
	ACK_Tool_At_WORK:= CMD_Tool_To_WORK AND Tool_At_WORK.0;
	ACK_Tool_At_HOME:= CMD_Tool_To_HOME AND Tool_At_HOME.0;

	ACK_CylAtWORK_Grp1:= CMD_CylToWORK_Grp1 AND Tool_At_WORK.1;
	ACK_CylAtHOME_Grp1:= CMD_CylToHOME_Grp1 AND Tool_At_HOME.1;
	ACK_CylAtWORK_Grp2:= CMD_CylToWORK_Grp2 AND Tool_At_WORK.2;
	ACK_CylAtHOME_Grp2:= CMD_CylToHOME_Grp2 AND Tool_At_HOME.2;
	ACK_CylAtWORK_Grp3:= CMD_CylToWORK_Grp3 AND Tool_At_WORK.3;
	ACK_CylAtHOME_Grp3:= CMD_CylToHOME_Grp3 AND Tool_At_HOME.3;
	ACK_CylAtWORK_Grp4:= CMD_CylToWORK_Grp4 AND Tool_At_WORK.4;
	ACK_CylAtHOME_Grp4:= CMD_CylToHOME_Grp4 AND Tool_At_HOME.4;
	ACK_CylAtWORK_Grp5:= CMD_CylToWORK_Grp5 AND Tool_At_WORK.5;
	ACK_CylAtHOME_Grp5:= CMD_CylToHOME_Grp5 AND Tool_At_HOME.5;














(*end*)
END_ACTION

ACTION ValveBank1:
(*+++++++++++THIS AREA IS CUSTOM PER INSTALLATION AND WILL HAVE TO BE MODIFIED PER +++++++++++++*)
(*+++++++++++THIS AREA IS CUSTOM PER INSTALLATION AND WILL HAVE TO BE MODIFIED PER +++++++++++++*)
(*+++++++++++THIS AREA IS CUSTOM PER INSTALLATION AND WILL HAVE TO BE MODIFIED PER +++++++++++++*)

(*+++++++++++VALVE BANK 1 +++++++++++++*)
(*+++++++++++VALVE BANK 1 +++++++++++++*)
(*+++++++++++VALVE BANK 1 +++++++++++++*)


	(*Valve 1, A+B*)
	(*Clamp 1, 2, 3, 4*)
		Valve1FB
			(
			Enable_Motion:= Enable_Motion ,
			Enable_Latch:= TRUE,					(*Enabling Runs Valve as detent type (maintained solenoids*)
			Enable_SideA_PreCharge:= FALSE,		(*Enabling Turns Side A PreCharge Active, reset when Side B is energized in Auto*)
			Enable_SideB_PreCharge:= TRUE,		(*Enabling Turns Side B PreCharge Active, reset when Side A is energized in Auto*)
			PreCharge_Time:= T#0.1S,
			Enable_Auto_Commands:= Enable_Motion,
			Enable_Manual_Commands:= FALSE,
			In_Manual_SideA_Command:= FALSE,
			In_Manual_SideB_Command:= FALSE,
			SideA_Indicator:= FALSE,
			SideB_Indicator:= FALSE,
			TurnOn_SideA_SOL=> N100.Q.0,
			TurnOn_SideB_SOL=> N100.Q.1,
			TurnOn_SideA_Indicator=> ,
			TurnOn_SideB_Indicator=>
			 );
		Valve1FB.In_Auto_SideA_Command:= CMD_Tool_To_WORK OR CMD_CylToWORK_Grp1;
		Valve1FB.In_Auto_SideB_Command:= CMD_Tool_To_HOME OR CMD_CylToHOME_Grp1;


	(*Valve 2, A+B*)
	(*Pins 1, 2, 3, 4*)
		Valve2FB
			(
			Enable_Motion:= Enable_Motion ,
			Enable_Latch:= TRUE,					(*Enabling Runs Valve as detent type (maintained solenoids*)
			Enable_SideA_PreCharge:= FALSE,		(*Enabling Turns Side A PreCharge Active, reset when Side B is energized in Auto*)
			Enable_SideB_PreCharge:= FALSE,		(*Enabling Turns Side B PreCharge Active, reset when Side A is energized in Auto*)
			PreCharge_Time:= T#0.10S,
			Enable_Auto_Commands:= Enable_Motion,
			Enable_Manual_Commands:= FALSE,
			In_Manual_SideA_Command:= FALSE,
			In_Manual_SideB_Command:= FALSE,
			SideA_Indicator:= FALSE,
			SideB_Indicator:= FALSE,
			TurnOn_SideA_SOL=> N100.Q.2,
			TurnOn_SideB_SOL=> N100.Q.3,
			TurnOn_SideA_Indicator=> ,
			TurnOn_SideB_Indicator=>
			 );
		Valve2FB.In_Auto_SideA_Command:= (*CMD_Tool_To_WORK OR*) CMD_CylToWORK_Grp2;
		Valve2FB.In_Auto_SideB_Command:= (*CMD_Tool_To_HOME OR*) CMD_CylToHOME_Grp2;


	(*Valve 3, A+B*)
	(*spare*)
		Valve3FB
			(
			Enable_Motion:= Enable_Motion ,
			Enable_Latch:= TRUE,				(*Enabling Runs Valve as detent type (maintained solenoids*)
			Enable_SideA_PreCharge:= FALSE,		(*Enabling Turns Side A PreCharge Active, reset when Side B is energized in Auto*)
			Enable_SideB_PreCharge:= FALSE,		(*Enabling Turns Side B PreCharge Active, reset when Side A is energized in Auto*)
			PreCharge_Time:= T#0.10S,
			Enable_Auto_Commands:= Enable_Motion,
			Enable_Manual_Commands:= FALSE,
			In_Manual_SideA_Command:= FALSE,
			In_Manual_SideB_Command:= FALSE,
			SideA_Indicator:= N100.Q.4,
			SideB_Indicator:= FALSE,
			TurnOn_SideA_SOL=> N100.Q.4,
			TurnOn_SideB_SOL=> N100.Q.5,
			TurnOn_SideA_Indicator=> ,
			TurnOn_SideB_Indicator=>
			 );
		Valve3FB.In_Auto_SideA_Command:= FALSE;
		Valve3FB.In_Auto_SideB_Command:= FALSE;


	(*Valve 4, A+B*)
	(*spare*)
		Valve4FB
			(
			Enable_Motion:= Enable_Motion ,
			Enable_Latch:= TRUE,					(*Enabling Runs Valve as detent type (maintained solenoids*)
			Enable_SideA_PreCharge:= FALSE,		(*Enabling Turns Side A PreCharge Active, reset when Side B is energized in Auto*)
			Enable_SideB_PreCharge:= FALSE,		(*Enabling Turns Side B PreCharge Active, reset when Side A is energized in Auto*)
			PreCharge_Time:= T#0.10S,
			Enable_Auto_Commands:= Enable_Motion,
			Enable_Manual_Commands:= FALSE,
			In_Manual_SideA_Command:= FALSE,
			In_Manual_SideB_Command:= FALSE,
			SideA_Indicator:= FALSE,
			SideB_Indicator:= FALSE,
			TurnOn_SideA_SOL=> N100.Q.6,
			TurnOn_SideB_SOL=> N100.Q.7,
			TurnOn_SideA_Indicator=> ,
			TurnOn_SideB_Indicator=>
			 );
		Valve4FB.In_Auto_SideA_Command:= FALSE;
		Valve4FB.In_Auto_SideB_Command:= FALSE;


	(*Valve 5, A+B*)
	(*spare*)
		Valve5FB
			(
			Enable_Motion:= Enable_Motion ,
			Enable_Latch:= TRUE,					(*Enabling Runs Valve as detent type (maintained solenoids*)
			Enable_SideA_PreCharge:= FALSE,		(*Enabling Turns Side A PreCharge Active, reset when Side B is energized in Auto*)
			Enable_SideB_PreCharge:= FALSE,		(*Enabling Turns Side B PreCharge Active, reset when Side A is energized in Auto*)
			PreCharge_Time:= T#0.10S,
			Enable_Auto_Commands:= Enable_Motion,
			Enable_Manual_Commands:= FALSE,
			In_Manual_SideA_Command:= FALSE,
			In_Manual_SideB_Command:= FALSE,
			SideA_Indicator:= FALSE,
			SideB_Indicator:= FALSE,
			TurnOn_SideA_SOL=> N100.Q.8,
			TurnOn_SideB_SOL=> N100.Q.9,
			TurnOn_SideA_Indicator=> ,
			TurnOn_SideB_Indicator=>
			 );
		Valve5FB.In_Auto_SideA_Command:= FALSE;
		Valve5FB.In_Auto_SideB_Command:= FALSE;


	(*Valve 6, A+B*)
	(*spare*)
		Valve6FB
			(
			Enable_Motion:= Enable_Motion ,
			Enable_Latch:= TRUE,					(*Enabling Runs Valve as detent type (maintained solenoids*)
			Enable_SideA_PreCharge:= FALSE,		(*Enabling Turns Side A PreCharge Active, reset when Side B is energized in Auto*)
			Enable_SideB_PreCharge:= FALSE,		(*Enabling Turns Side B PreCharge Active, reset when Side A is energized in Auto*)
			PreCharge_Time:= T#0.10S,
			Enable_Auto_Commands:= Enable_Motion,
			Enable_Manual_Commands:= FALSE,
			In_Manual_SideA_Command:= FALSE,
			In_Manual_SideB_Command:= FALSE,
			SideA_Indicator:= FALSE,
			SideB_Indicator:= FALSE,
			TurnOn_SideA_SOL=> N100.Q.10,
			TurnOn_SideB_SOL=> N100.Q.11,
			TurnOn_SideA_Indicator=> ,
			TurnOn_SideB_Indicator=>
			 );
		Valve6FB.In_Auto_SideA_Command:= FALSE;
		Valve6FB.In_Auto_SideB_Command:= FALSE;


	(*Valve 7, A+B*)
	(*spare*)
		Valve7FB
			(
			Enable_Motion:= Enable_Motion ,
			Enable_Latch:= TRUE,					(*Enabling Runs Valve as detent type (maintained solenoids*)
			Enable_SideA_PreCharge:= FALSE,		(*Enabling Turns Side A PreCharge Active, reset when Side B is energized in Auto*)
			Enable_SideB_PreCharge:= FALSE,		(*Enabling Turns Side B PreCharge Active, reset when Side A is energized in Auto*)
			PreCharge_Time:= T#0.10S,
			Enable_Auto_Commands:= Enable_Motion,
			Enable_Manual_Commands:= FALSE,
			In_Manual_SideA_Command:= FALSE,
			In_Manual_SideB_Command:= FALSE,
			SideA_Indicator:= FALSE,
			SideB_Indicator:= FALSE,
			TurnOn_SideA_SOL=> N100.Q.12,
			TurnOn_SideB_SOL=> N100.Q.13,
			TurnOn_SideA_Indicator=> ,
			TurnOn_SideB_Indicator=>
			 );
		Valve7FB.In_Auto_SideA_Command:= FALSE;
		Valve7FB.In_Auto_SideB_Command:= FALSE;


	(*Valve 8, A+B*)
	(*spare*)
		Valve8FB
			(
			Enable_Motion:= Enable_Motion ,
			Enable_Latch:= TRUE,					(*Enabling Runs Valve as detent type (maintained solenoids*)
			Enable_SideA_PreCharge:= FALSE,		(*Enabling Turns Side A PreCharge Active, reset when Side B is energized in Auto*)
			Enable_SideB_PreCharge:= FALSE,		(*Enabling Turns Side B PreCharge Active, reset when Side A is energized in Auto*)
			PreCharge_Time:= T#0.10S,
			Enable_Auto_Commands:= Enable_Motion,
			Enable_Manual_Commands:= FALSE,
			In_Manual_SideA_Command:= FALSE,
			In_Manual_SideB_Command:= FALSE,
			SideA_Indicator:= FALSE,
			SideB_Indicator:= FALSE,
			TurnOn_SideA_SOL=> N100.Q.14,
			TurnOn_SideB_SOL=> N100.Q.15,
			TurnOn_SideA_Indicator=> ,
			TurnOn_SideB_Indicator=>
			 );
		Valve8FB.In_Auto_SideA_Command:= FALSE;
		Valve8FB.In_Auto_SideB_Command:= FALSE;


	(*Valve 9, A+B*)
	(*spare*)
		Valve9FB
			(
			Enable_Motion:= Enable_Motion ,
			Enable_Latch:= TRUE,					(*Enabling Runs Valve as detent type (maintained solenoids*)
			Enable_SideA_PreCharge:= FALSE,		(*Enabling Turns Side A PreCharge Active, reset when Side B is energized in Auto*)
			Enable_SideB_PreCharge:= FALSE,		(*Enabling Turns Side B PreCharge Active, reset when Side A is energized in Auto*)
			PreCharge_Time:= T#0.10S,
			Enable_Auto_Commands:= Enable_Motion,
			Enable_Manual_Commands:= FALSE,
			In_Manual_SideA_Command:= FALSE,
			In_Manual_SideB_Command:= FALSE,
			SideA_Indicator:= FALSE,
			SideB_Indicator:= FALSE,
			TurnOn_SideA_SOL=> N100.Q.16,
			TurnOn_SideB_SOL=> N100.Q.17,
			TurnOn_SideA_Indicator=> ,
			TurnOn_SideB_Indicator=>
			 );
		Valve9FB.In_Auto_SideA_Command:= FALSE;
		Valve9FB.In_Auto_SideB_Command:= FALSE;


	(*Valve 10, A+B*)
	(*spare*)
		Valve10FB
			(
			Enable_Motion:= Enable_Motion ,
			Enable_Latch:= TRUE,					(*Enabling Runs Valve as detent type (maintained solenoids*)
			Enable_SideA_PreCharge:= FALSE,		(*Enabling Turns Side A PreCharge Active, reset when Side B is energized in Auto*)
			Enable_SideB_PreCharge:= FALSE,		(*Enabling Turns Side B PreCharge Active, reset when Side A is energized in Auto*)
			PreCharge_Time:= T#0.10S,
			Enable_Auto_Commands:= Enable_Motion,
			Enable_Manual_Commands:= FALSE,
			In_Manual_SideA_Command:= FALSE,
			In_Manual_SideB_Command:= FALSE,
			SideA_Indicator:= FALSE,
			SideB_Indicator:= FALSE,
			TurnOn_SideA_SOL=> N100.Q.18,
			TurnOn_SideB_SOL=> N100.Q.19,
			TurnOn_SideA_Indicator=> ,
			TurnOn_SideB_Indicator=>
			 );
		Valve10FB.In_Auto_SideA_Command:= FALSE;
		Valve10FB.In_Auto_SideB_Command:= FALSE;


	(*Valve 11, A+B*)
	(*spare*)
		Valve11FB
			(
			Enable_Motion:= Enable_Motion ,
			Enable_Latch:= TRUE,					(*Enabling Runs Valve as detent type (maintained solenoids*)
			Enable_SideA_PreCharge:= FALSE,		(*Enabling Turns Side A PreCharge Active, reset when Side B is energized in Auto*)
			Enable_SideB_PreCharge:= FALSE,		(*Enabling Turns Side B PreCharge Active, reset when Side A is energized in Auto*)
			PreCharge_Time:= T#0.10S,
			Enable_Auto_Commands:= Enable_Motion,
			Enable_Manual_Commands:= FALSE,
			In_Manual_SideA_Command:= FALSE,
			In_Manual_SideB_Command:= FALSE,
			SideA_Indicator:= FALSE,
			SideB_Indicator:= FALSE,
			TurnOn_SideA_SOL=> N100.Q.20,
			TurnOn_SideB_SOL=> N100.Q.21,
			TurnOn_SideA_Indicator=> ,
			TurnOn_SideB_Indicator=>
			 );
		Valve11FB.In_Auto_SideA_Command:= FALSE;
		Valve11FB.In_Auto_SideB_Command:= FALSE;


	(*Valve 12, A+B*)
	(*spare*)
		Valve12FB
			(
			Enable_Motion:= Enable_Motion ,
			Enable_Latch:= TRUE,					(*Enabling Runs Valve as detent type (maintained solenoids*)
			Enable_SideA_PreCharge:= FALSE,		(*Enabling Turns Side A PreCharge Active, reset when Side B is energized in Auto*)
			Enable_SideB_PreCharge:= FALSE,		(*Enabling Turns Side B PreCharge Active, reset when Side A is energized in Auto*)
			PreCharge_Time:= T#0.10S,
			Enable_Auto_Commands:= Enable_Motion,
			Enable_Manual_Commands:= FALSE,
			In_Manual_SideA_Command:= FALSE,
			In_Manual_SideB_Command:= FALSE,
			SideA_Indicator:= FALSE,
			SideB_Indicator:= FALSE,
			TurnOn_SideA_SOL=> N100.Q.22,
			TurnOn_SideB_SOL=> N100.Q.23,
			TurnOn_SideA_Indicator=> ,
			TurnOn_SideB_Indicator=>
			 );
		Valve12FB.In_Auto_SideA_Command:= FALSE;
		Valve12FB.In_Auto_SideB_Command:= FALSE;


	(*Valve 13, A+B*)
	(*spare*)
		Valve13FB
			(
			Enable_Motion:= Enable_Motion ,
			Enable_Latch:= TRUE,					(*Enabling Runs Valve as detent type (maintained solenoids*)
			Enable_SideA_PreCharge:= FALSE,		(*Enabling Turns Side A PreCharge Active, reset when Side B is energized in Auto*)
			Enable_SideB_PreCharge:= FALSE,		(*Enabling Turns Side B PreCharge Active, reset when Side A is energized in Auto*)
			PreCharge_Time:= T#0.10S,
			Enable_Auto_Commands:= Enable_Motion,
			Enable_Manual_Commands:= FALSE,
			In_Manual_SideA_Command:= FALSE,
			In_Manual_SideB_Command:= FALSE,
			SideA_Indicator:= FALSE,
			SideB_Indicator:= FALSE,
			TurnOn_SideA_SOL=> N100.Q.24,
			TurnOn_SideB_SOL=> N100.Q.25,
			TurnOn_SideA_Indicator=> ,
			TurnOn_SideB_Indicator=>
			 );
		Valve13FB.In_Auto_SideA_Command:= FALSE;
		Valve13FB.In_Auto_SideB_Command:= FALSE;


	(*Valve 14, A+B*)
	(*spare*)
		Valve14FB
			(
			Enable_Motion:= Enable_Motion ,
			Enable_Latch:= TRUE,					(*Enabling Runs Valve as detent type (maintained solenoids*)
			Enable_SideA_PreCharge:= FALSE,		(*Enabling Turns Side A PreCharge Active, reset when Side B is energized in Auto*)
			Enable_SideB_PreCharge:= FALSE,		(*Enabling Turns Side B PreCharge Active, reset when Side A is energized in Auto*)
			PreCharge_Time:= T#0.10S,
			Enable_Auto_Commands:= Enable_Motion,
			Enable_Manual_Commands:= FALSE,
			In_Manual_SideA_Command:= FALSE,
			In_Manual_SideB_Command:= FALSE,
			SideA_Indicator:= FALSE,
			SideB_Indicator:= FALSE,
			TurnOn_SideA_SOL=> N100.Q.26,
			TurnOn_SideB_SOL=> N100.Q.27,
			TurnOn_SideA_Indicator=> ,
			TurnOn_SideB_Indicator=>
			 );
		Valve14FB.In_Auto_SideA_Command:= FALSE;
		Valve14FB.In_Auto_SideB_Command:= FALSE;


	(*Valve 15, A+B*)
	(*spare*)
		Valve15FB
			(
			Enable_Motion:= Enable_Motion ,
			Enable_Latch:= TRUE,					(*Enabling Runs Valve as detent type (maintained solenoids*)
			Enable_SideA_PreCharge:= FALSE,		(*Enabling Turns Side A PreCharge Active, reset when Side B is energized in Auto*)
			Enable_SideB_PreCharge:= FALSE,		(*Enabling Turns Side B PreCharge Active, reset when Side A is energized in Auto*)
			PreCharge_Time:= T#0.10S,
			Enable_Auto_Commands:= Enable_Motion,
			Enable_Manual_Commands:= FALSE,
			In_Manual_SideA_Command:= FALSE,
			In_Manual_SideB_Command:= FALSE,
			SideA_Indicator:= FALSE,
			SideB_Indicator:= FALSE,
			TurnOn_SideA_SOL=> N100.Q.28,
			TurnOn_SideB_SOL=> N100.Q.29,
			TurnOn_SideA_Indicator=> ,
			TurnOn_SideB_Indicator=>
			 );
		Valve15FB.In_Auto_SideA_Command:= FALSE;
		Valve15FB.In_Auto_SideB_Command:= FALSE;


	(*Valve 16, A+B*)
	(*spare*)
		Valve16FB
			(
			Enable_Motion:= Enable_Motion ,
			Enable_Latch:= TRUE,					(*Enabling Runs Valve as detent type (maintained solenoids*)
			Enable_SideA_PreCharge:= FALSE,		(*Enabling Turns Side A PreCharge Active, reset when Side B is energized in Auto*)
			Enable_SideB_PreCharge:= FALSE,		(*Enabling Turns Side B PreCharge Active, reset when Side A is energized in Auto*)
			PreCharge_Time:= T#0.10S,
			Enable_Auto_Commands:= Enable_Motion,
			Enable_Manual_Commands:= FALSE,
			In_Manual_SideA_Command:= FALSE,
			In_Manual_SideB_Command:= FALSE,
			SideA_Indicator:= FALSE,
			SideB_Indicator:= FALSE,
			TurnOn_SideA_SOL=> N100.Q.30,
			TurnOn_SideB_SOL=> N100.Q.31,
			TurnOn_SideA_Indicator=> ,
			TurnOn_SideB_Indicator=>
			 );
		Valve16FB.In_Auto_SideA_Command:= FALSE;
		Valve16FB.In_Auto_SideB_Command:= FALSE;


























(*end*)
END_ACTION

ACTION Xfer_To_UI:
	(*Transfer General Status and I/O Images for Display On HMI*)
	Discrete_Image.CLFaults1:= CLFaults1;
	Discrete_Image.CLFaults2:= CLFaults2;
	Discrete_Image.CLFaults3:= CLFaults3;
	Discrete_Image.CLFaults4:= CLFaults4;
	Discrete_Image.CLFaulted:= CLFaulted;
	Discrete_Image.PPFaults:= PPFaults;
	Discrete_Image.PPFaulted:= PPFaulted;

	Discrete_Image.N01:=N01;
	Discrete_Image.N02:=N02;
	Discrete_Image.N03:=N03;
	Discrete_Image.N04:=N04;
	Discrete_Image.N05:=N05;
	Discrete_Image.N06:=N06;
	Discrete_Image.N07:=N07;
	Discrete_Image.N08:=N08;
	Discrete_Image.N09:=N09;
	Discrete_Image.N100:=N100;
	Discrete_Image.N100_STAT:=N100_STAT;
	Discrete_Image.NodeLayout:=NodeLayout;
	Discrete_Image.NodeState:=NodeState;

	Discrete_Image.ID:= ID;
	Discrete_Image.ECatSlave_Cable_Breaks:= ECatSlave_Cable_Breaks;
	Discrete_Image.Input_Node_Count:= Input_Node_Count;
	Discrete_Image.VB_Node_Count:= VB_Node_Count;
















(*end*)
END_ACTION

END_PROGRAM

// ---- POUs/Misc/Servo_Motion.TcPOU
PROGRAM Servo_Motion
VAR
(*Servo Drives*)
			SD: ARRAY[0..30] OF  FB_GTAC_ServoSystem_20211214;
			IC_LoopIndex: UINT;
			SD_LoopIndex: UINT;
			Axis_LoopIndex: UINT;
			
			IC_Requesting_LocalControl: UDINT;
			SD_Requested: UDINT;
			Axis_Requested: UDINT;
			Axis2_Requested: UDINT;
			In_Local_Control: BOOL;
			Local_Control_Stop: ARRAY [0..2] OF BOOL;
			

END_VAR

(*--------------------------------------- Service Common Servo Drive Requests from UI(s) ------------------------------------------------*)

	Handle_LocalControl_Requests();


(*------------------------------------ Setup Individual Servo Drive Data -------------------------------*)
(* DEBUG, EXAMPLE ONLY*)

(*Servo Drive 1*)
(*Axis1 = add axis description here*)
(*Axis2 = add axis description here*)
	(*Inputs*)
	SD[1].FB_In.Enable_Motion[1]:= MAIN.Control_Power_ON										(*DEBUG, remove FALSE and add in other code as required to enable drive, blt*)
								OR TRUE;
	SD[1].FB_In.Enable_Motion[2]:= MAIN.Control_Power_ON										(*DEBUG, remove FALSE and add in other code as required to enable drive, blt*)
								OR TRUE;
	SD[1].FB_In.ECAT_AmsID:= MAIN.ECAT_Master.AmsID;
	SD[1].FB_In.Prev_EcatNode_Present:= NOT MAIN.IS01.EK1100_NotPresent; 						(*Ensure Previous Node Exists to determine Ecat Cable Break of this Devices Input Cable*)
	SD[1].FB_In.Teach_Enable[1]:= TRUE;															(*Set Input to true to allow UI teaching of servo, set to false to hard code program positional data*)
	SD[1].FB_In.Teach_Enable[2]:= TRUE;															(*Set Input to true to allow UI teaching of servo, set to false to hard code program positional data*)
	SD[1].FB_In.Axis_Common_Name[1]:= 'add axis 1 name here';
	SD[1].FB_In.Axis_Common_Name[2]:= 'add axis 2 name here';
	SD[1].FB_In.Option_Type:= 0;																(*0=AX5xxx type, 10=EL72xx type*)
	SD[1].FB_In.Option_Axis_Count:= 2; 															(*Min 1, Max 2*)
	SD[1].FB_In.Axis_Is_Absolute[1]:= FALSE;
	SD[1].FB_In.Axis_Is_Absolute[2]:= FALSE;
	
	SD[1].FB_In.Home_Position_Switch[1]:= TRUE;												(*Map Home Position Verification Switch here/Axis*)
	SD[1].FB_In.Quick_Home_REQ[1]:= FALSE;													(*Alternate Request to Directly Home axis - Specify homing type below*)
	SD[1].FB_In.Homing_Type[1]:= MC_DefaultHoming;											(*Non-Delayed Home Request Type Select*)
	SD[1].FB_In.Homing_Offset[1]:= 0.0;														(*Value of Reference position when homed*)
	SD[1].FB_In.Home_Position_Switch[2]:= TRUE;												(*Map Home Position Verification Switch here/Axis*)
	SD[1].FB_In.Quick_Home_REQ[2]:= FALSE;													(*Alternate Request to home axis  - Specify homing type below*)
	SD[1].FB_In.Homing_Type[2]:= MC_DefaultHoming;											(*Non-Delayed Home Request Type Select*)
	SD[1].FB_In.Homing_Offset[2]:= 0.0;														(*Value of Reference position when homed*)

	SD[1].FB_In.Soft_Limit_Max[1]:=1000;															(*Set Axis1 Pos Software Limit here*)
	SD[1].FB_In.Soft_Limit_Min[1]:= -1000;															(*Set Axis1 Neg Software Limit here*)
	SD[1].FB_In.Soft_Limit_Max[2]:= 1000;															(*Set Axis2 Pos Software Limit here*)
	SD[1].FB_In.Soft_Limit_Min[2]:= -1000;															(*Set Axis2 Neg Software Limit here*)
	SD[1].FB_In.Disable_Soft_Limits[1]:= FALSE;													(*Allow this Axis to run without softlimits*)
	SD[1].FB_In.Disable_Soft_Limits[2]:= FALSE;													(*Allow this Axis to run without softlimits*)

	SD[1].FB_In.Max_Torque[1]:= 1000;															(*Axis1 Maximum Torque, Eg: 1000 = 100.0%, 800 = 80.0%*)
	SD[1].FB_In.Max_Torque[2]:= 1000;															(*Axis1 Maximum Torque, Eg. 1000 = 100.0%, 800 = 80.0%*)
	SD[1].FB_In.System_Max_Velocity[1]:= 8733;													(*Must be set per System / Axis (find maximum velcity value in Config)*)
	SD[1].FB_In.System_Max_Velocity[2]:= 1500;													(*Must be set per System / Axis (find maximum velcity value in Config)*)

	SD[1].FB_In.MicroInch_Value[1]:=0.1;															(*Value Servo Will Micro Inch*)
	SD[1].FB_In.MicroInch_Value[2]:=0.1;															(*Value Servo Will Micro Inch*)
	SD[1].FB_In.Error_Reset[1]:= In_From_ICxx.ControlPower1 OR MAIN.Starting_Scan_Pulse;			(*Will handle all levels of faults*)
	SD[1].FB_In.Error_Reset[2]:= In_From_ICxx.ControlPower1 OR MAIN.Starting_Scan_Pulse;			(*Will handle all levels of faults*)
	SD[1].FB_In.Program_Reset[1]:= FALSE;														(*Map Requirements for full program reset here*)
	SD[1].FB_In.Program_Reset[2]:= FALSE;														(*Map Requirements for full program reset here*)
	SD[1].FB_In.PlayBack_StepPermit[1]:= TRUE;													(*Map process interlocks here to halt playback at each step*)
	SD[1].FB_In.PlayBack_StepPermit[2]:= TRUE;													(*Map process interlocks here to halt playback at each step*)
	(*Last Call on Stopping Motion*)
	SD[1].FB_In.Stop_PlayBack[1]:= Local_Control_Stop[1] OR FALSE;										(*Stop All Playback, add custom application stop requirements instad of False*)
	SD[1].FB_In.Stop_PlayBack[2]:= Local_Control_Stop[2] OR FALSE;										(*Stop All Playback, add custom application stop requirements instad of False*)


	(*EXAMPLE ONLY of explicit step call type of motion, programmed motion can be done as well*)
(*
	(*Override Playback Mode Inputs Here with Higher Level Commands*)
	IF Fix101.In_Manual AND NOT In_Local_Control AND SD[1].Homed[1] AND SD[1].Homed[2]
		THEN
			SD[1].FB_In.Mode_Select[1]:= 2;
			SD[1].FB_In.Mode_Select[2]:= 2;
			SD[1].FB_In.Stop_PlayBack[1]:= NOT SD[1].FB_In.Start_Explicit_StepCall[1];
			SD[1].FB_In.Stop_PlayBack[2]:= NOT SD[1].FB_In.Start_Explicit_StepCall[2];
		IF Fix101.OP103_Data.Home_REQ AND Fix101.OP103_Data.Tool_At_Position.30
			THEN
			SD[1].FB_In.Explicit_Step_REQ[1]:= 1;
		END_IF;
			SD[1].FB_In.Start_Explicit_StepCall[1]:= Fix101.OP103_Data.Home_REQ AND SD[1].FB_In.Explicit_Step_REQ[1]=1;
		IF Fix101.OP104_Data.Home_REQ AND Fix101.OP103_Data.Tool_At_Position.30
									AND Fix101.OP104_Data.Tool_At_Position.29
			THEN
			SD[1].FB_In.Explicit_Step_REQ[2]:= 1;
		END_IF;
			SD[1].FB_In.Start_Explicit_StepCall[2]:= Fix101.OP104_Data.Home_REQ AND SD[1].FB_In.Explicit_Step_REQ[2]=1;
	END_IF;
	IF Fix101.In_Auto
		THEN
		(*Play Mode Inputs*)
		SD[1].FB_In.Mode_Select[1]:= 1;
		SD[1].FB_In.Mode_Select[2]:= 1;
		SD[1].FB_In.PlayBack_Speed_Percentage[1]:= 100;											(*Set Auto Playback Speed Here*)
		SD[1].FB_In.PlayBack_Speed_Percentage[2]:= 100;											(*Set Auto Playback Speed Here*)
		(*Set Playback Here Axis 1*)
			SD[1].FB_In.Start_Explicit_StepCall[1]:= (Fix101.OP103_DataPers.Step_Complete.0 AND NOT Fix101.OP103_DataPers.Step_Complete.1 AND Fix101.OP110_Data.Interlocks_ToNext.29 AND (SD[1].FB_In.Explicit_Step_REQ[1] = 2))
												OR (Fix101.OP103_DataPers.Step_Complete.6 AND NOT Fix101.OP103_DataPers.Step_Complete.7 AND (SD[1].FB_In.Explicit_Step_REQ[1] = 1));
				IF Fix101.OP103_DataPers.Step_Complete.0 AND NOT Fix101.OP103_DataPers.Step_Complete.1 AND Fix101.OP110_Data.Interlocks_ToNext.29
					THEN
					SD[1].FB_In.Explicit_Step_REQ[1]:= 2;
				ELSIF Fix101.OP103_DataPers.Step_Complete.6 AND NOT Fix101.OP103_DataPers.Step_Complete.7
					THEN
					SD[1].FB_In.Explicit_Step_REQ[1]:= 1;
				ELSE
					SD[1].FB_In.Explicit_Step_REQ[1]:= 0;
				END_IF;

		(*Set Playback Here Axis 2*)
			SD[1].FB_In.Start_Explicit_StepCall[2]:= (Fix101.OP104_DataPers.Step_Complete.1 AND NOT Fix101.OP104_DataPers.Step_Complete.2 AND (SD[1].FB_In.Explicit_Step_REQ[2] = Fix101.Model_ID + 10))
												OR  (Fix101.OP104_DataPers.Step_Complete.5 AND NOT Fix101.OP104_DataPers.Step_Complete.6 AND (SD[1].FB_In.Explicit_Step_REQ[2] = 1));
				IF Fix101.OP104_DataPers.Step_Complete.1 AND NOT Fix101.OP104_DataPers.Step_Complete.2
					THEN
					SD[1].FB_In.Explicit_Step_REQ[2]:= Fix101.Model_ID + 10;
				ELSIF Fix101.OP104_DataPers.Step_Complete.5 AND NOT Fix101.OP104_DataPers.Step_Complete.6
					THEN
					SD[1].FB_In.Explicit_Step_REQ[2]:= 1;
				ELSE
					SD[1].FB_In.Explicit_Step_REQ[2]:= 0;
				END_IF;


			SD[1].FB_In.Start_PlayBack[1]:= FALSE;
			SD[1].FB_In.Start_PlayBack[2]:= FALSE;
			(*Map process interlocks here to halt playback at each step*)
			SD[1].FB_In.PlayBack_StepPermit[1]:= TRUE;
			SD[1].FB_In.PlayBack_StepPermit[2]:= TRUE;
	END_IF;
*)
	(*Call actual FB*)
	SD[1]();
	
	(*Output Data*)
	Out_To_ICxx.SD[1].Discrete_Image:= SD[1].Discrete_Image;
	Out_To_ICxx.SD[1].ECAT_Cable_Breaks:= SD[1].ECatSlave_Cable_Breaks;

ACTION Handle_LocalControl_Requests:
(*DEBUG, Brent working on this during TcUI Migration, this will require more testing, blt*)
(*DEBUG, need to finalize local control code, REQS and ACKS added to UI udts, blt*)

(*------------------------------------------- Handle Local Control Requests from UI ---------------------------------------*)

(*Set some default values upon machine bootup*)
	IF MAIN.Starting_Scan_Pulse
		THEN
		FOR SD_LoopIndex:= 1 TO GTAC_CONFIG.Option_SD_Count DO

		In_From_ICxx.SD[SD_LoopIndex].PlayBack_Speed_Percentage[1]:= 50;	 (*Set default playback speed to 50% of maximum system velocity*)
		In_From_ICxx.SD[SD_LoopIndex].PlayBack_Speed_Percentage[2]:= 50;	 (*Set default playback speed to 50% of maximum system velocity*)
		In_From_ICxx.SD[SD_LoopIndex].Teach_Params[1].Velocity:= 25;		(*Set default playback speed to 25% of maximum system velocity*)
		In_From_ICxx.SD[SD_LoopIndex].Teach_Params[2].Velocity:= 25;		(*Set default playback speed to 25% of maximum system velocity*)
		In_From_ICxx.SD[SD_LoopIndex].Teach_Params[1].Accel:= 5000;
		In_From_ICxx.SD[SD_LoopIndex].Teach_Params[1].Decel:= 5000;
		In_From_ICxx.SD[SD_LoopIndex].Teach_Params[2].Accel:= 5000;
		In_From_ICxx.SD[SD_LoopIndex].Teach_Params[2].Decel:= 5000;
		END_FOR;
	END_IF;

(*First Blank All Requests Regardless*)
		FOR SD_LoopIndex:= 1 TO GTAC_CONFIG.Option_SD_Count DO
			SD[SD_LoopIndex].FB_In.Explicit_Step_REQ[1]:= 0;
			SD[SD_LoopIndex].FB_In.Explicit_Step_REQ[2]:= 0;
			SD[SD_LoopIndex].FB_In.Start_Explicit_StepCall[1]:= FALSE;
			SD[SD_LoopIndex].FB_In.Start_Explicit_StepCall[2]:= FALSE;
			SD[SD_LoopIndex].FB_In.Start_PlayBack[1]:= FALSE;
			SD[SD_LoopIndex].FB_In.Start_PlayBack[2]:= FALSE;
			SD[SD_LoopIndex].FB_In.Stop_PlayBack[1]:= FALSE;
			SD[SD_LoopIndex].FB_In.Stop_PlayBack[2]:= FALSE;

			(*Teach Mode Inputs*)
			SD[SD_LoopIndex].FB_In.Teach_Servo_HomePos[1]:= FALSE;
			SD[SD_LoopIndex].FB_In.Teach_Servo_HomePos[2]:= FALSE;
			SD[SD_LoopIndex].FB_In.Teach_JogFast_Plus[1]:= FALSE;
			SD[SD_LoopIndex].FB_In.Teach_JogFast_Plus[2]:= FALSE;
			SD[SD_LoopIndex].FB_In.Teach_JogFast_Minus[1]:= FALSE;
			SD[SD_LoopIndex].FB_In.Teach_JogFast_Minus[2]:= FALSE;
			SD[SD_LoopIndex].FB_In.Teach_JogSlow_Plus[1]:= FALSE;
			SD[SD_LoopIndex].FB_In.Teach_JogSlow_Plus[2]:= FALSE;
			SD[SD_LoopIndex].FB_In.Teach_JogSlow_Minus[1]:= FALSE;
			SD[SD_LoopIndex].FB_In.Teach_JogSlow_Minus[2]:= FALSE;
			SD[SD_LoopIndex].FB_In.Teach_Inch_Plus[1]:= FALSE;
			SD[SD_LoopIndex].FB_In.Teach_Inch_Plus[2]:= FALSE;
			SD[SD_LoopIndex].FB_In.Teach_Inch_Minus[1]:= FALSE;
			SD[SD_LoopIndex].FB_In.Teach_Inch_Minus[2]:= FALSE;
			SD[SD_LoopIndex].FB_In.Teach_MicroInch_Enable[1]:= FALSE;
			SD[SD_LoopIndex].FB_In.Teach_MicroInch_Enable[2]:= FALSE;
			SD[SD_LoopIndex].FB_In.Teach_Record_CurrentPos[1]:= FALSE;
			SD[SD_LoopIndex].FB_In.Teach_Record_CurrentPos[2]:= FALSE;
			SD[SD_LoopIndex].FB_In.Teach_ParamsOverwrite_Flag[1]:= FALSE;
			SD[SD_LoopIndex].FB_In.Teach_ParamsOverwrite_Flag[2]:= FALSE;
		END_FOR;

		
		

(*Transfer User Requests to Specific Servo System*)
	FOR SD_LoopIndex:= 1 TO GTAC_CONFIG.Option_SD_Count DO
		(*Handle Local Control Requests from UI(s)*)
		Out_To_ICxx.SD[SD_LoopIndex].AxisLocalControl_IC_ACKS:= In_From_ICxx.SD[SD_LoopIndex].AxisLocalControl_IC_REQS;		
		FOR Axis_LoopIndex:= 1 TO 2 DO
			IF (Out_To_ICxx.SD[SD_LoopIndex].AxisLocalControl_IC_ACKS[Axis_LoopIndex] >0) AND (Out_To_ICxx.SD[SD_LoopIndex].AxisLocalControl_IC_ACKS[Axis_LoopIndex] < GTAC_Config.Option_IC_Count)
				THEN

				
				(*Mode Select*)
				SD[SD_LoopIndex].FB_In.Mode_Select[Axis_LoopIndex]:= In_From_ICxx.SD[SD_LoopIndex].Mode_Select[Axis_LoopIndex];
	
				(*Play Mode Inputs*)
				SD[SD_LoopIndex].FB_In.PlayBack_Speed_Percentage[Axis_LoopIndex]:= In_From_ICxx.SD[SD_LoopIndex].PlayBack_Speed_Percentage[Axis_LoopIndex];
				SD[SD_LoopIndex].FB_In.Explicit_Step_REQ[Axis_LoopIndex]:= In_From_ICxx.SD[SD_LoopIndex].Explicit_Step_REQ[Axis_LoopIndex];
				SD[SD_LoopIndex].FB_In.Start_Explicit_StepCall[Axis_LoopIndex]:= In_From_ICxx.SD[SD_LoopIndex].Start_Explicit_StepCall[Axis_LoopIndex];
				SD[SD_LoopIndex].FB_In.Start_PlayBack[Axis_LoopIndex]:= In_From_ICxx.SD[SD_LoopIndex].Start_PlayBack[Axis_LoopIndex];
				Local_Control_Stop[Axis_LoopIndex]:= In_From_ICxx.SD[SD_LoopIndex].Stop_PlayBack[Axis_LoopIndex] OR In_From_ICxx.Cycle_Hold;
	
				(*Teach Mode Inputs*)
				SD[SD_LoopIndex].FB_In.Teach_Params[Axis_LoopIndex]:= In_From_ICxx.SD[SD_LoopIndex].Teach_Params[Axis_LoopIndex];
				SD[SD_LoopIndex].FB_In.Teach_JogFast_Plus[Axis_LoopIndex]:= In_From_ICxx.SD[SD_LoopIndex].Teach_JogFast_Plus[Axis_LoopIndex];
				SD[SD_LoopIndex].FB_In.Teach_JogFast_Minus[Axis_LoopIndex]:= In_From_ICxx.SD[SD_LoopIndex].Teach_JogFast_Minus[Axis_LoopIndex];
				SD[SD_LoopIndex].FB_In.Teach_JogSlow_Plus[Axis_LoopIndex]:= In_From_ICxx.SD[SD_LoopIndex].Teach_JogSlow_Plus[Axis_LoopIndex];
				SD[SD_LoopIndex].FB_In.Teach_JogSlow_Minus[Axis_LoopIndex]:= In_From_ICxx.SD[SD_LoopIndex].Teach_JogSlow_Minus[Axis_LoopIndex];
				SD[SD_LoopIndex].FB_In.Teach_Inch_Plus[Axis_LoopIndex]:= In_From_ICxx.SD[SD_LoopIndex].Teach_Inch_Plus[Axis_LoopIndex];
				SD[SD_LoopIndex].FB_In.Teach_Inch_Minus[Axis_LoopIndex]:= In_From_ICxx.SD[SD_LoopIndex].Teach_Inch_Minus[Axis_LoopIndex];
				SD[SD_LoopIndex].FB_In.Teach_MicroInch_Enable[Axis_LoopIndex]:= In_From_ICxx.SD[SD_LoopIndex].Teach_MicroInch_Enable[Axis_LoopIndex];
				SD[SD_LoopIndex].FB_In.Teach_Record_CurrentPos[Axis_LoopIndex]:= In_From_ICxx.SD[SD_LoopIndex].Teach_Record_CurrentPos[Axis_LoopIndex];
				SD[SD_LoopIndex].FB_In.Teach_ParamsOverwrite_Flag[Axis_LoopIndex]:= In_From_ICxx.SD[SD_LoopIndex].Teach_ParamsOverwrite_Flag[Axis_LoopIndex];
					 (*Requires home Position Switch to be on and performs an MC_Direct Home when Callibrate Button is pushed for 5 seconds - Also see Quick_Home_REQ in Servo_Motion as an alternate type of homing*)
					SD[SD_LoopIndex].FB_In.Teach_Servo_HomePos[Axis_LoopIndex]:= In_From_ICxx.SD[SD_LoopIndex].Teach_Servo_HomePos[Axis_LoopIndex];
			END_IF;
		END_FOR;
	END_FOR;
END_ACTION

END_PROGRAM

// ---- POUs/FBs/FB_GTAC_ServoSystem_20211214.TcPOU
(*
FB for use with a simple single axis "robot" can be combined for multi axis control:
(Originally designed for use with EL72xx series servo terminals but may be adopted for other controllers that use type "Axis_Ref" as IN/OUT interface)
Original Author(S): Brent Lekx-Toniolo OF Sodecia GTAC;
**NOTE: Re-created for use a FB for a Servo Drive, therefore multi axis can be supported by a single drive.
------------------------------------------------------------------------------------------
	REVISION NOTES:
	Date: Jan 2015
	- initial concept: b.lekx-toniolo

	Date: Aug 2015
	- Modifications for restart: r.remillard	

	Date: Sep 2015
	- Modifications for Jog Function
	- Added Velocity and Acc to Jog fast and Jog slow

	Date: Feb 17 2016
	- added extenal program reset bit, JVD
	- added fb_Drive_Stop.Execute to Manual jog logic to prevent an error being generated if the drive is being told to stop, JVD

	Version 20160805
		- Modified for full selectable use with EL7xxx series terminals and AX5xxx series drives including dual axis support, b.lekx-toniolo
		- Re-created interface for use with index image concept (for endless extensibility), b.lekx-toniolo
	Version 20161124
		- Seperated out Enable Motion for Each Axis, b.lekx-toniolo
	Version 20161214
		- Added In_Start_Position Flags, b.lekx-toniolo
		- Added Software Limit Inputs, b.lekx-toniolo
		- Added Home Position Inputs, b.lekx-toniolo

	Version 20180731
		- Added teach enable function, b.donnell
		- Added ability to directly enter positional data, velocity, accel, decel, motion type and end flag for each position, b.donnell
		- Added Teach_Enable state to the discrete image to the screen, b.donnell
		- Added the ability to home the servo while it is in Auto, b.donnell
		- Added MoveModulo function to the FB and brokeout FB into some actions, b.donnell
	Version 20191001
		- Added In_Standstill and In_Stopping reads, j.underhill & b.lekx-toniolo
		- Added In-Standstill to over-all ReadyFor_Motion, j.underhill & b.lekx-toniolo
	Version20200609
		- Update Instance OF FB_AX5805_Info, d.silva / j.underhill / b.lekx-toniolo
		- Passed Value OF Axis count TO new the above, d.silva / j.underhill / b.lekx-toniolo
	Version 20211214
		- Updates to allow input of Reference Position from outside of FB (GH issue 67), c.drees / b.lekx-toniolo
		- Updates for better possible reset of AX5805 upon error (GH issue 65), c.drees / b.lekx-toniolo
------------------------------------------------------------------------------------------
*)
FUNCTION_BLOCK FB_GTAC_ServoSystem_20211214
VAR_INPUT
	Enable_FB: BOOL;
	FB_In: udt_Generic_ServoDrive_FBIN_20211214;
	Corrected_Position: ARRAY[0..2] OF LREAL;
END_VAR
VAR
	///EBUS Power Restoration, may or may not be used
	T01 AT %I*: udt_EL94xx;
	///Servo Terminal
	T03 AT %I*: udt_EL7211_20150115;
	///AX5000 Series Nodes
	Drive AT %I*: udt_AX5206_20160804;
	Drive_AX5805 AT %I*: udt_AX5805_20160804;
	Drive_AX5805_Reset AT %Q*: BOOL;
	Drive_BipolarTorque AT %Q*: ARRAY[0..2] OF INT ;
	FB_AX5805_Info: FB_Ax5805_GetInfo_20200609;
	/// AX5xxx Series Axis Diag and Reset 
	FB_Axis_Diag: ARRAY[0..2] OF FB_AxisDiag_20160810;
	ST_AX5000_Diag: ARRAY[0..2] OF udt_AX5000Diag;
	ResetReq: ARRAY[0..2] OF BOOL;
	DiagReq: ARRAY[0..2] OF BOOL;
	ResetAct: ARRAY[0..2] OF BOOL;
	DiagAct: ARRAY[0..2] OF BOOL;
	/// Nodes States
	DiscreteNode_OK: BOOL;
	///Cable Break States
	ECatSlave_Cable_Breaks: UDINT;
	///Coupler is Not Present on Bus when expected
	Drive_NotPresent: BOOL;
	///Port B of AX5xxx is OUT
	AX5xxx_PortB_MissingLink: BOOL;
	///Port D of AX5xxx is Safety Slot
	AX5xxx_PortD_MissingLink: BOOL;
	///Axis Array Index
	Axis_Index: INT;
	///Develop data Area for Interface with the Axis
	Axis: ARRAY[0..2] OF Axis_REF;
	///Develop Instances (array types for mulit axis use)
	fb_Power: ARRAY[0..2] OF MC_Power;
	fb_Move_Abs: ARRAY[0..2] OF MC_MoveAbsolute;
	fb_Move_Vel: ARRAY[0..2] OF MC_MoveVelocity;
	fb_Move_Add: ARRAY[0..2] OF MC_MoveAdditive;
	fb_Move_Mod: ARRAY[0..2] OF MC_MoveModulo;
	fb_Jog: ARRAY[0..2] OF MC_Jog;
	fb_Move_AbsTeach: ARRAY[0..2] OF MC_MoveAbsolute;
	fb_Stop: ARRAY[0..2] OF MC_Stop;
	fb_Set_Position: ARRAY[0..2] OF MC_SetPosition;
	fb_Set_Home: ARRAY[0..2] OF MC_Home;
	fb_SetBool_EnPosMax: ARRAY[0..2] OF MC_WriteBoolParameter;
	fb_SetBool_EnPosMin: ARRAY[0..2] OF MC_WriteBoolParameter;
	fb_Set_PosMax: ARRAY[0..2] OF MC_WriteParameter;
	fb_Set_PosMin: ARRAY[0..2] OF MC_WriteParameter;
	fb_ReadBool_EnPosMax: ARRAY[0..2] OF MC_ReadBoolParameter;
	fb_ReadBool_EnPosMin: ARRAY[0..2] OF MC_ReadBoolParameter;
	Type_MC_AxisParameter: MC_AxisParameter;
	fb_Reset: ARRAY[0..2] OF MC_Reset;
	fb_SoE_Reset: ARRAY[0..2] OF FB_SoEReset;
	fb_Actual_Position: ARRAY[0..2] OF MC_ReadActualPosition;
	fb_Read_Status: ARRAY[0..2] OF MC_ReadStatus;
	///General Internals
	In_Play: ARRAY[0..2] OF BOOL;
	In_Teach: ARRAY[0..2] OF BOOL;
	Auto_Run: ARRAY[0..2] OF BOOL;
	Auto_Velocity: ARRAY[0..2] OF LREAL;
	Auto_Accel: ARRAY[0..2] OF LREAL;
	Auto_Decel: ARRAY[0..2] OF LREAL;
	Manual_Velocity: ARRAY[0..2] OF LREAL;
	Manual_Accel: ARRAY[0..2] OF LREAL;
	Manual_Decel: ARRAY[0..2] OF LREAL;
	Manual_Distance: ARRAY[0..2] OF LREAL;
	///Timer for Setting of Home Position
	SET_HomeTMR: ARRAY[0..2] OF TON;
	///Timer To Delay Servo Drive Commands Until Enable Has Been Achieved
	Auto_ABS_DelayTMR: ARRAY[0..2] OF TON;
	///Inching Variable
	Inching_Value: ARRAY[0..2] OF REAL;
	///Misc
	RPulse: ARRAY[0..10] OF R_TRIG;
END_VAR
VAR PERSISTENT
	///Stored (Taught) Postional Data (IE Programmed Points)
	Program_Positions: ARRAY[0..2] OF ARRAY[0..15] OF udt_SingleAxis_MoveData_20160908;
	Current_Step_Pointer: ARRAY[0..2] OF UINT;
	Step_Running: ARRAY[0..2] OF BOOL;
	Program_Running: ARRAY[0..2] OF BOOL;
	Program_Complete: ARRAY[0..2] OF BOOL;
	Step_Complete: ARRAY[0..2] OF BOOL;
	test: BOOL;
END_VAR
VAR_OUTPUT
	FB_Ok: BOOL;
	In_Play_ACK: ARRAY[0..2] OF BOOL;
	In_Teach_ACK: ARRAY[0..2] OF BOOL;
	Readyfor_Motion: ARRAY[0..2] OF BOOL;
	Readyfor_TeachMotion: ARRAY[0..2] OF BOOL;
	In_Error: ARRAY[0..2] OF BOOL;
	Error_ID: ARRAY[0..2] OF UDINT;
	Homed: ARRAY[0..2] OF BOOL;
	In_Requested_Position: ARRAY[0..2] OF BOOL;
	In_Standstill: ARRAY[0..2] OF BOOL;
	In_Stopping: ARRAY[0..2] OF BOOL;
	In_Motion: ARRAY[0..2] OF BOOL;
	At_Current_Step: ARRAY[0..2] OF UINT;
	Cycle_Complete: ARRAY[0..2] OF BOOL;
	Current_Position: ARRAY[0..2] OF LREAL;
	Discrete_Image: udt_Drive_Image_20190816;
END_VAR

(*Set FB_OK to True*)
		FB_OK:= TRUE;
(*Set Boundries*)
IF FB_In.Option_Axis_Count>2
	THEN FB_In.Option_Axis_Count:=2;
ELSIF FB_In.Option_Axis_Count<1
	THEN FB_In.Option_Axis_Count:=1;
ELSIF FB_In.Option_Type=10
	THEN FB_In.Option_Axis_Count:=1;
END_IF;


(*$$$$$$$$$$$$$$$$$$$$$$$$$$$$$$$$$$$$$$$$$$$$$$$$Gather Status Of Hardware $$$$$$$$$$$$$$$$$$$$$$$$$$$$$$$$$$$$$$$$$$$$$$$$$$$$*)
(*Discrete I/O Nodes*)
	IF FB_In.Option_Type=0 AND (Drive.InfoData.State=8)
		AND (Drive_AX5805.InfoData.State=8)
		THEN
			DiscreteNode_OK:=TRUE;
	ELSIF FB_In.Option_Type=10 AND (T01.InfoData.State=8)
		AND (T03.InfoData.State=8)
		THEN
			DiscreteNode_OK:=TRUE;
	ELSE
			DiscreteNode_OK:=FALSE;

	END_IF;

(*EtherCAT Cable Break Detection*)
	(*Develop Port Connection Warning Flags*)
	IF Drive.InfoData.State=257  (*State Machine for Slave Not Present*)
		THEN Drive_NotPresent:= TRUE;
	ELSE Drive_NotPresent := FALSE;
	END_IF;

	IF Drive.InfoData.State=16#2408 (*State Machine for Link Missing at Port B*)
		THEN AX5xxx_PortB_MissingLink:= TRUE; (*PortB is X5 Port*)
	ELSE AX5xxx_PortB_MissingLink := FALSE;
	END_IF;

	IF Drive.InfoData.State=17416 (*State Machine for Link Missing at Port D*)
		THEN AX5xxx_PortD_MissingLink:= TRUE; (*PortD is Safety Slot*)
	ELSE AX5xxx_PortD_MissingLink := FALSE;
	END_IF;

	(*Wrap up break Flags to Variable for shipment to UI*)
	ECatSlave_Cable_Breaks.0:= Drive_NotPresent AND FB_In.Prev_EcatNode_Present;
	ECatSlave_Cable_Breaks.1:= AX5xxx_PortB_MissingLink; (*X5 Out Port Warning*)
	ECatSlave_Cable_Breaks.4:= AX5xxx_PortD_MissingLink; (*Warning for AX5805 (safety slot)*)
	ECatSlave_Cable_Breaks.16:= Discrete_Image.Drive_C1D_ErrorStruct[1].bFeedbackError
								OR Discrete_Image.Axis_ErrorID[1]=16#4550;			(*Warning for Axis1 Motor Cable*)
	ECatSlave_Cable_Breaks.17:= Discrete_Image.Drive_C1D_ErrorStruct[2].bFeedbackError
								OR Discrete_Image.Axis_ErrorID[2]=16#4550;			(*Warning for Axis2 Motor Cable*)


(*Get AX5805 Status*)
	(*Inputs to FB*)
	FB_Ax5805_Info.Ecat_Master_AmsNetID:= FB_In.ECAT_AmsID;
	FB_Ax5805_Info.Axis_Count:= FB_In.Option_Axis_Count;

	(*Call actual FB*)
	FB_AX5805_Info(AX5805_InfoData:= Drive_AX5805.InfoData);


(*all items past this point are indexed via Axis Index*)
FOR Axis_Index:= 1 TO FB_In.Option_Axis_Count
	DO
	(*Get Status*)
		fb_Read_Status[Axis_Index].Enable:= TRUE;
		fb_Read_Status[Axis_Index](Axis:= Axis[Axis_Index]);
	(*Get Servo Drive Data*)
		(*Get Current Position*)
		fb_Actual_Position[Axis_Index].Enable:= TRUE;
		fb_Actual_Position[Axis_Index](Axis:= Axis[Axis_Index]);


(*$$$$$$$$$$$$$$$$$$$$$$$$$$$$$$$$$$$$$$$$$$$$$$$$ Internal Code $$$$$$$$$$$$$$$$$$$$$$$$$$$$$$$$$$$$$$$$$$$$$$$$$$$$$$$$$$$$$$$$$$$$*)
(*Ensure Postion Data zero is always blank*)
	Program_Positions[Axis_Index][0].Position:= 0;
	Program_Positions[Axis_Index][0].Velocity:= 0;
	Program_Positions[Axis_Index][0].Accel:= 0;
	Program_Positions[Axis_Index][0].Decel:= 0;
	Program_Positions[Axis_Index][0].Move_Type:= 0;
	Program_Positions[Axis_Index][0].End_Flag:= 0;

(*Auto / Manual Mode Code*)
	IF FB_In.Mode_Select[Axis_Index].0 AND NOT FB_In.Mode_Select[Axis_Index].1
		THEN
			In_Play[Axis_Index]:= TRUE;
	END_IF;
	IF NOT FB_In.Mode_Select[Axis_Index].0 AND FB_In.Mode_Select[Axis_Index].1
		THEN
			In_Play[Axis_Index]:= FALSE;
	END_IF;
	In_Teach[Axis_Index]:= NOT In_Play[Axis_Index];


(*%%%%%%%%%%%%%%%%%%%%%%%%%%%%% General Enable of Axis %%%%%%%%%%%%%%%%%%%%%%%%*)

	(*Handle General Stop*)
	IF FB_In.Enable_Motion[Axis_Index] AND NOT FB_In.Stop_PlayBack[Axis_Index]
		THEN
			fb_Stop[Axis_Index].Execute:= FALSE;
	ELSIF (NOT FB_In.Enable_Motion[Axis_Index] AND fb_Power[Axis_Index].Enable) OR FB_In.Stop_PlayBack[Axis_Index]
		THEN
			fb_Move_VEL[Axis_Index].Execute:= FALSE;
			fb_Move_ABS[Axis_Index].Execute:= FALSE;
			fb_Move_MOD[Axis_Index].Execute:= FALSE;
			IF FB_In.System_Stop_Decel[Axis_Index] <> 0
				THEN
				fb_Stop[Axis_Index].Deceleration:= Fb_In.System_Stop_Decel[Axis_Index]; (*Set User Entered Decel*)
			ELSE
				fb_Stop[Axis_Index].Deceleration:= FB_In.System_Max_Velocity[Axis_Index]*10; (*Decel Default*)
			END_IF;
			fb_Stop[Axis_Index].Execute:= TRUE;

	END_IF;

	(*Handle General Enable*)
	IF FB_In.Enable_Motion[Axis_Index]
		THEN
		(*Drive Enable and Override*)
		fb_Power[Axis_Index].Enable:= TRUE;
		fb_Power[Axis_Index].Enable_Negative:= TRUE;
		fb_Power[Axis_Index].Enable_Positive:= TRUE;
		fb_Power[Axis_Index].Override:= 100;
	ELSIF NOT FB_In.Enable_Motion[Axis_Index] AND fb_Stop[Axis_Index].Done 	(*Once all Absolute Moves are stopped and/or completed then disable Drive*)
		THEN
		fb_Power[Axis_Index].Enable:= FALSE;
		fb_Power[Axis_Index].Enable_Negative:= FALSE;
		fb_Power[Axis_Index].Enable_Positive:= FALSE;
		fb_Power[Axis_Index].Override:= 0;
	END_IF;

	(*Handle Software Limits*)
	(*Load Read fbs*)
	fb_ReadBool_EnPosMax[Axis_Index].ParameterNumber:= AxisEnMaxSoftPosLimit;
	fb_ReadBool_EnPosMax[Axis_Index].ReadMode:= READMODE_CYCLIC;
	fb_ReadBool_EnPosMax[Axis_Index].Enable:= TRUE;
	fb_ReadBool_EnPosMax[Axis_Index](Axis:= Axis[Axis_Index]);
	fb_ReadBool_EnPosMin[Axis_Index].ParameterNumber:= AxisEnMinSoftPosLimit;
	fb_ReadBool_EnPosMin[Axis_Index].ReadMode:= READMODE_CYCLIC;
	fb_ReadBool_EnPosMin[Axis_Index].Enable:= TRUE;
	fb_ReadBool_EnPosMin[Axis_Index](Axis:= Axis[Axis_Index]);

	(*Enable or Disable Softlimits depending on state of Homed*)
	(*If Axis is not callibrated, and user is not requesting, remove software limits*)
	IF NOT Homed[Axis_Index] AND NOT FB_IN.Teach_Servo_HomePos[Axis_Index] OR (FB_In.Disable_Soft_Limits[Axis_Index] )
		AND ((fb_ReadBool_EnPosMax[Axis_Index].Value = TRUE) OR (fb_ReadBool_EnPosMin[Axis_Index].Value = TRUE))
		AND NOT fb_SetBool_EnPosMin[Axis_Index].Done
		THEN
		fb_SetBool_EnPosMax[Axis_Index].ParameterNumber:= AxisEnMaxSoftPosLimit;
		fb_SetBool_EnPosMax[Axis_Index].Value:= FALSE;
		fb_SetBool_EnPosMax[Axis_Index].Execute:= TRUE;
		fb_SetBool_EnPosMax[Axis_Index](Axis:= Axis[Axis_Index]);

		fb_Set_PosMax[Axis_Index].ParameterNumber:= AxisMaxSoftPosLimit;
		fb_Set_PosMax[Axis_Index].Value:= 0;
		fb_Set_PosMax[Axis_Index].Execute:= TRUE;
		fb_Set_PosMax[Axis_Index](Axis:= Axis[Axis_Index]);

		fb_SetBool_EnPosMin[Axis_Index].ParameterNumber:= AxisEnMinSoftPosLimit;
		fb_SetBool_EnPosMin[Axis_Index].Value:= FALSE;
		fb_SetBool_EnPosMin[Axis_Index].Execute:= TRUE;
		fb_SetBool_EnPosMin[Axis_Index](Axis:= Axis[Axis_Index]);

		fb_Set_PosMin[Axis_Index].ParameterNumber:= AxisMinSoftPosLimit;
		fb_Set_PosMin[Axis_Index].Value:= 0;
		fb_Set_PosMin[Axis_Index].Execute:= TRUE;
		fb_Set_PosMin[Axis_Index](Axis:= Axis[Axis_Index]);

	ELSIF Homed[Axis_Index] AND NOT FB_In.Disable_Soft_Limits[Axis_Index]
		AND ((fb_ReadBool_EnPosMax[Axis_Index].Value = FALSE) OR (fb_ReadBool_EnPosMin[Axis_Index].Value = FALSE))
		AND NOT fb_SetBool_EnPosMin[Axis_Index].Done
		THEN
		fb_SetBool_EnPosMax[Axis_Index].ParameterNumber:= AxisEnMaxSoftPosLimit;
		fb_SetBool_EnPosMax[Axis_Index].Value:= TRUE;
		fb_SetBool_EnPosMax[Axis_Index].Execute:= TRUE;
		fb_SetBool_EnPosMax[Axis_Index](Axis:= Axis[Axis_Index]);

		fb_Set_PosMax[Axis_Index].ParameterNumber:= AxisMaxSoftPosLimit;
		fb_Set_PosMax[Axis_Index].Value:= FB_In.Soft_Limit_Max[Axis_Index];
		fb_Set_PosMax[Axis_Index].Execute:= TRUE;
		fb_Set_PosMax[Axis_Index](Axis:= Axis[Axis_Index]);

		fb_SetBool_EnPosMin[Axis_Index].ParameterNumber:= AxisEnMinSoftPosLimit;
		fb_SetBool_EnPosMin[Axis_Index].Value:= TRUE;
		fb_SetBool_EnPosMin[Axis_Index].Execute:= TRUE;
		fb_SetBool_EnPosMin[Axis_Index](Axis:= Axis[Axis_Index]);

		fb_Set_PosMin[Axis_Index].ParameterNumber:= AxisMinSoftPosLimit;
		fb_Set_PosMin[Axis_Index].Value:= FB_In.Soft_Limit_Min[Axis_Index];
		fb_Set_PosMin[Axis_Index].Execute:= TRUE;
		fb_Set_PosMin[Axis_Index](Axis:= Axis[Axis_Index]);
	ELSE
		fb_SetBool_EnPosMax[Axis_Index].Execute:= FALSE;
		fb_SetBool_EnPosMin[Axis_Index].Execute:= FALSE;
		fb_Set_PosMax[Axis_Index].Execute:= FALSE;
		fb_Set_PosMin[Axis_Index].Execute:= FALSE;

	END_IF;




(*General Set-Up Parameters/Function calls for Servo Drive*)
		fb_Power[Axis_Index](Axis:= Axis[Axis_Index]);
		fb_Stop[Axis_Index](Axis:=Axis[Axis_Index]);

(*~~~~~~~~~~~~~~~~~~~~~~~~~~~~~~~~~~~~~~~ Auto Cycle Code ~~~~~~~~~~~~~~~~~~~~~~~~~~~~~~~~~~~*)

(*Action Calls*)
Teach_Mode();
Move_Absolute();
Move_Modulo();
Move_Velocity();


	(*If Teach_Enable is not true, you cannot teach an axis position from the screen, must be hardcoded with values below - initialized in Servo_Motion*)
		IF NOT FB_in.Teach_Enable[1] AND FB_In.Rotary_Axis[1]
			THEN
			(*Axis 1 Position, Velocity, Accel, Decel, Motion Type and End Flag for each program position*)
				Program_Positions[1][0].Position:= FB_In.Position[1][0];
				Program_Positions[1][1].Position:= FB_In.Position[1][1];
				Program_Positions[1][2].Position:= FB_In.Position[1][2];
				Program_Positions[1][3].Position:= FB_In.Position[1][3];
				Program_Positions[1][4].Position:= FB_In.Position[1][4];
				Program_Positions[1][5].Position:= FB_In.Position[1][5];
				Program_Positions[1][6].Position:= FB_In.Position[1][6];
				Program_Positions[1][7].Position:= FB_In.Position[1][7];
				Program_Positions[1][8].Position:= FB_In.Position[1][8];
				Program_Positions[1][9].Position:= FB_In.Position[1][9];
				Program_Positions[1][10].Position:= FB_In.Position[1][10];
				Program_Positions[1][11].Position:= FB_In.Position[1][11];
				Program_Positions[1][12].Position:= FB_In.Position[1][12];
				Program_Positions[1][13].Position:= FB_In.Position[1][13];
				Program_Positions[1][14].Position:= FB_In.Position[1][14];
				Program_Positions[1][15].Position:= FB_In.Position[1][15];

				Program_Positions[1][0].Velocity:= FB_In.Auto_Vel[1][0];
				Program_Positions[1][1].Velocity:= FB_In.Auto_Vel[1][1];
				Program_Positions[1][2].Velocity:= FB_In.Auto_Vel[1][2];
				Program_Positions[1][3].Velocity:= FB_In.Auto_Vel[1][3];
				Program_Positions[1][4].Velocity:= FB_In.Auto_Vel[1][4];
				Program_Positions[1][5].Velocity:= FB_In.Auto_Vel[1][5];
				Program_Positions[1][6].Velocity:= FB_In.Auto_Vel[1][6];
				Program_Positions[1][7].Velocity:= FB_In.Auto_Vel[1][7];
				Program_Positions[1][8].Velocity:= FB_In.Auto_Vel[1][8];
				Program_Positions[1][9].Velocity:= FB_In.Auto_Vel[1][9];
				Program_Positions[1][10].Velocity:= FB_In.Auto_Vel[1][10];
				Program_Positions[1][11].Velocity:= FB_In.Auto_Vel[1][11];
				Program_Positions[1][12].Velocity:= FB_In.Auto_Vel[1][12];
				Program_Positions[1][13].Velocity:= FB_In.Auto_Vel[1][13];
				Program_Positions[1][14].Velocity:= FB_In.Auto_Vel[1][14];
				Program_Positions[1][15].Velocity:= FB_In.Auto_Vel[1][15];

				Program_Positions[1][0].Accel:= FB_In.Auto_Accel[1][0];
				Program_Positions[1][1].Accel:= FB_In.Auto_Accel[1][1];
				Program_Positions[1][2].Accel:= FB_In.Auto_Accel[1][2];
				Program_Positions[1][3].Accel:= FB_In.Auto_Accel[1][3];
				Program_Positions[1][4].Accel:= FB_In.Auto_Accel[1][4];
				Program_Positions[1][5].Accel:= FB_In.Auto_Accel[1][5];
				Program_Positions[1][6].Accel:= FB_In.Auto_Accel[1][6];
				Program_Positions[1][7].Accel:= FB_In.Auto_Accel[1][7];
				Program_Positions[1][8].Accel:= FB_In.Auto_Accel[1][8];
				Program_Positions[1][9].Accel:= FB_In.Auto_Accel[1][9];
				Program_Positions[1][10].Accel:= FB_In.Auto_Accel[1][10];
				Program_Positions[1][11].Accel:= FB_In.Auto_Accel[1][11];
				Program_Positions[1][12].Accel:= FB_In.Auto_Accel[1][12];
				Program_Positions[1][13].Accel:= FB_In.Auto_Accel[1][13];
				Program_Positions[1][14].Accel:= FB_In.Auto_Accel[1][14];
				Program_Positions[1][15].Accel:= FB_In.Auto_Accel[1][15];

				Program_Positions[1][0].Decel:= FB_In.Auto_Decel[1][0];
				Program_Positions[1][1].Decel:= FB_In.Auto_Decel[1][1];
				Program_Positions[1][2].Decel:= FB_In.Auto_Decel[1][2];
				Program_Positions[1][3].Decel:= FB_In.Auto_Decel[1][3];
				Program_Positions[1][4].Decel:= FB_In.Auto_Decel[1][4];
				Program_Positions[1][5].Decel:= FB_In.Auto_Decel[1][5];
				Program_Positions[1][6].Decel:= FB_In.Auto_Decel[1][6];
				Program_Positions[1][7].Decel:= FB_In.Auto_Decel[1][7];
				Program_Positions[1][8].Decel:= FB_In.Auto_Decel[1][8];
				Program_Positions[1][9].Decel:= FB_In.Auto_Decel[1][9];
				Program_Positions[1][10].Decel:= FB_In.Auto_Decel[1][10];
				Program_Positions[1][11].Decel:= FB_In.Auto_Decel[1][11];
				Program_Positions[1][12].Decel:= FB_In.Auto_Decel[1][12];
				Program_Positions[1][13].Decel:= FB_In.Auto_Decel[1][13];
				Program_Positions[1][14].Decel:= FB_In.Auto_Decel[1][14];
				Program_Positions[1][15].Decel:= FB_In.Auto_Decel[1][15];

				Program_Positions[1][0].End_Flag:= FB_In.Auto_EndFlag[1][0];
				Program_Positions[1][1].End_Flag:= FB_In.Auto_EndFlag[1][1];
				Program_Positions[1][2].End_Flag:= FB_In.Auto_EndFlag[1][2];
				Program_Positions[1][3].End_Flag:= FB_In.Auto_EndFlag[1][3];
				Program_Positions[1][4].End_Flag:= FB_In.Auto_EndFlag[1][4];
				Program_Positions[1][5].End_Flag:= FB_In.Auto_EndFlag[1][5];
				Program_Positions[1][6].End_Flag:= FB_In.Auto_EndFlag[1][6];
				Program_Positions[1][7].End_Flag:= FB_In.Auto_EndFlag[1][7];
				Program_Positions[1][8].End_Flag:= FB_In.Auto_EndFlag[1][8];
				Program_Positions[1][9].End_Flag:= FB_In.Auto_EndFlag[1][9];
				Program_Positions[1][10].End_Flag:= FB_In.Auto_EndFlag[1][10];
				Program_Positions[1][11].End_Flag:= FB_In.Auto_EndFlag[1][11];
				Program_Positions[1][12].End_Flag:= FB_In.Auto_EndFlag[1][12];
				Program_Positions[1][13].End_Flag:= FB_In.Auto_EndFlag[1][13];
				Program_Positions[1][14].End_Flag:= FB_In.Auto_EndFlag[1][14];
				Program_Positions[1][15].End_Flag:= FB_In.Auto_EndFlag[1][15];

				Program_Positions[1][0].Move_Type:= FB_In.Auto_MoveType[1][0];
				Program_Positions[1][1].Move_Type:= FB_In.Auto_MoveType[1][1];
				Program_Positions[1][2].Move_Type:= FB_In.Auto_MoveType[1][2];
				Program_Positions[1][3].Move_Type:= FB_In.Auto_MoveType[1][3];
				Program_Positions[1][4].Move_Type:= FB_In.Auto_MoveType[1][4];
				Program_Positions[1][5].Move_Type:= FB_In.Auto_MoveType[1][5];
				Program_Positions[1][6].Move_Type:= FB_In.Auto_MoveType[1][6];
				Program_Positions[1][7].Move_Type:= FB_In.Auto_MoveType[1][7];
				Program_Positions[1][8].Move_Type:= FB_In.Auto_MoveType[1][8];
				Program_Positions[1][9].Move_Type:= FB_In.Auto_MoveType[1][9];
				Program_Positions[1][10].Move_Type:= FB_In.Auto_MoveType[1][10];
				Program_Positions[1][11].Move_Type:= FB_In.Auto_MoveType[1][11];
				Program_Positions[1][12].Move_Type:= FB_In.Auto_MoveType[1][12];
				Program_Positions[1][13].Move_Type:= FB_In.Auto_MoveType[1][13];
				Program_Positions[1][14].Move_Type:= FB_In.Auto_MoveType[1][14];
				Program_Positions[1][15].Move_Type:= FB_In.Auto_MoveType[1][15];

		END_IF;

		IF NOT FB_in.Teach_Enable[2] AND FB_In.Rotary_Axis[2]
			THEN
			(*Axis 2 Position, Velocity, Accel, Decel, Motion Type and End Flag for each program position*)
				Program_Positions[2][0].Position:= FB_In.Position[2][0];
				Program_Positions[2][1].Position:= FB_In.Position[2][1];
				Program_Positions[2][2].Position:= FB_In.Position[2][2];
				Program_Positions[2][3].Position:= FB_In.Position[2][3];
				Program_Positions[2][4].Position:= FB_In.Position[2][4];
				Program_Positions[2][5].Position:= FB_In.Position[2][5];
				Program_Positions[2][6].Position:= FB_In.Position[2][6];
				Program_Positions[2][7].Position:= FB_In.Position[2][7];
				Program_Positions[2][8].Position:= FB_In.Position[2][8];
				Program_Positions[2][9].Position:= FB_In.Position[2][9];
				Program_Positions[2][10].Position:= FB_In.Position[2][10];
				Program_Positions[2][11].Position:= FB_In.Position[2][11];
				Program_Positions[2][12].Position:= FB_In.Position[2][12];
				Program_Positions[2][13].Position:= FB_In.Position[2][13];
				Program_Positions[2][14].Position:= FB_In.Position[2][14];
				Program_Positions[2][15].Position:= FB_In.Position[2][15];

				Program_Positions[2][0].Velocity:= FB_In.Auto_Vel[2][0];
				Program_Positions[2][1].Velocity:= FB_In.Auto_Vel[2][1];
				Program_Positions[2][2].Velocity:= FB_In.Auto_Vel[2][2];
				Program_Positions[2][3].Velocity:= FB_In.Auto_Vel[2][3];
				Program_Positions[2][4].Velocity:= FB_In.Auto_Vel[2][4];
				Program_Positions[2][5].Velocity:= FB_In.Auto_Vel[2][5];
				Program_Positions[2][6].Velocity:= FB_In.Auto_Vel[2][6];
				Program_Positions[2][7].Velocity:= FB_In.Auto_Vel[2][7];
				Program_Positions[2][8].Velocity:= FB_In.Auto_Vel[2][8];
				Program_Positions[2][9].Velocity:= FB_In.Auto_Vel[2][9];
				Program_Positions[2][10].Velocity:= FB_In.Auto_Vel[2][10];
				Program_Positions[2][11].Velocity:= FB_In.Auto_Vel[2][11];
				Program_Positions[2][12].Velocity:= FB_In.Auto_Vel[2][12];
				Program_Positions[2][13].Velocity:= FB_In.Auto_Vel[2][13];
				Program_Positions[2][14].Velocity:= FB_In.Auto_Vel[2][14];
				Program_Positions[2][15].Velocity:= FB_In.Auto_Vel[2][15];

				Program_Positions[2][0].Accel:= FB_In.Auto_Accel[2][0];
				Program_Positions[2][1].Accel:= FB_In.Auto_Accel[2][1];
				Program_Positions[2][2].Accel:= FB_In.Auto_Accel[2][2];
				Program_Positions[2][3].Accel:= FB_In.Auto_Accel[2][3];
				Program_Positions[2][4].Accel:= FB_In.Auto_Accel[2][4];
				Program_Positions[2][5].Accel:= FB_In.Auto_Accel[2][5];
				Program_Positions[2][6].Accel:= FB_In.Auto_Accel[2][6];
				Program_Positions[2][7].Accel:= FB_In.Auto_Accel[2][7];
				Program_Positions[2][8].Accel:= FB_In.Auto_Accel[2][8];
				Program_Positions[2][9].Accel:= FB_In.Auto_Accel[2][9];
				Program_Positions[2][10].Accel:= FB_In.Auto_Accel[2][10];
				Program_Positions[2][11].Accel:= FB_In.Auto_Accel[2][11];
				Program_Positions[2][12].Accel:= FB_In.Auto_Accel[2][12];
				Program_Positions[2][13].Accel:= FB_In.Auto_Accel[2][13];
				Program_Positions[2][14].Accel:= FB_In.Auto_Accel[2][14];
				Program_Positions[2][15].Accel:= FB_In.Auto_Accel[2][15];

				Program_Positions[2][0].Decel:= FB_In.Auto_Decel[2][0];
				Program_Positions[2][1].Decel:= FB_In.Auto_Decel[2][1];
				Program_Positions[2][2].Decel:= FB_In.Auto_Decel[2][2];
				Program_Positions[2][3].Decel:= FB_In.Auto_Decel[2][3];
				Program_Positions[2][4].Decel:= FB_In.Auto_Decel[2][4];
				Program_Positions[2][5].Decel:= FB_In.Auto_Decel[2][5];
				Program_Positions[2][6].Decel:= FB_In.Auto_Decel[2][6];
				Program_Positions[2][7].Decel:= FB_In.Auto_Decel[2][7];
				Program_Positions[2][8].Decel:= FB_In.Auto_Decel[2][8];
				Program_Positions[2][9].Decel:= FB_In.Auto_Decel[2][9];
				Program_Positions[2][10].Decel:= FB_In.Auto_Decel[2][10];
				Program_Positions[2][11].Decel:= FB_In.Auto_Decel[2][11];
				Program_Positions[2][12].Decel:= FB_In.Auto_Decel[2][12];
				Program_Positions[2][13].Decel:= FB_In.Auto_Decel[2][13];
				Program_Positions[2][14].Decel:= FB_In.Auto_Decel[2][14];
				Program_Positions[2][15].Decel:= FB_In.Auto_Decel[2][15];

				Program_Positions[2][0].End_Flag:= FB_In.Auto_EndFlag[2][0];
				Program_Positions[2][1].End_Flag:= FB_In.Auto_EndFlag[2][1];
				Program_Positions[2][2].End_Flag:= FB_In.Auto_EndFlag[2][2];
				Program_Positions[2][3].End_Flag:= FB_In.Auto_EndFlag[2][3];
				Program_Positions[2][4].End_Flag:= FB_In.Auto_EndFlag[2][4];
				Program_Positions[2][5].End_Flag:= FB_In.Auto_EndFlag[2][5];
				Program_Positions[2][6].End_Flag:= FB_In.Auto_EndFlag[2][6];
				Program_Positions[2][7].End_Flag:= FB_In.Auto_EndFlag[2][7];
				Program_Positions[2][8].End_Flag:= FB_In.Auto_EndFlag[2][8];
				Program_Positions[2][9].End_Flag:= FB_In.Auto_EndFlag[2][9];
				Program_Positions[2][10].End_Flag:= FB_In.Auto_EndFlag[2][10];
				Program_Positions[2][11].End_Flag:= FB_In.Auto_EndFlag[2][11];
				Program_Positions[2][12].End_Flag:= FB_In.Auto_EndFlag[2][12];
				Program_Positions[2][13].End_Flag:= FB_In.Auto_EndFlag[2][13];
				Program_Positions[2][14].End_Flag:= FB_In.Auto_EndFlag[2][14];
				Program_Positions[2][15].End_Flag:= FB_In.Auto_EndFlag[2][15];

				Program_Positions[2][0].Move_Type:= FB_In.Auto_MoveType[2][0];
				Program_Positions[2][1].Move_Type:= FB_In.Auto_MoveType[2][1];
				Program_Positions[2][2].Move_Type:= FB_In.Auto_MoveType[2][2];
				Program_Positions[2][3].Move_Type:= FB_In.Auto_MoveType[2][3];
				Program_Positions[2][4].Move_Type:= FB_In.Auto_MoveType[2][4];
				Program_Positions[2][5].Move_Type:= FB_In.Auto_MoveType[2][5];
				Program_Positions[2][6].Move_Type:= FB_In.Auto_MoveType[2][6];
				Program_Positions[2][7].Move_Type:= FB_In.Auto_MoveType[2][7];
				Program_Positions[2][8].Move_Type:= FB_In.Auto_MoveType[2][8];
				Program_Positions[2][9].Move_Type:= FB_In.Auto_MoveType[2][9];
				Program_Positions[2][10].Move_Type:= FB_In.Auto_MoveType[2][10];
				Program_Positions[2][11].Move_Type:= FB_In.Auto_MoveType[2][11];
				Program_Positions[2][12].Move_Type:= FB_In.Auto_MoveType[2][12];
				Program_Positions[2][13].Move_Type:= FB_In.Auto_MoveType[2][13];
				Program_Positions[2][14].Move_Type:= FB_In.Auto_MoveType[2][14];
				Program_Positions[2][15].Move_Type:= FB_In.Auto_MoveType[2][15];
		END_IF;

(*################################################# Home Routine AUTO ###########################################*)

IF ReadyFor_Motion[Axis_Index] AND In_Play_ACK[Axis_Index] AND NOT FB_In.Stop_PlayBack[Axis_Index] AND NOT Cycle_Complete[Axis_Index]
	THEN

			(*Simple Direct, Delayed Homing Routine*)
			SET_HomeTMR[Axis_Index].IN:= FB_In.Enable_Motion[Axis_Index] AND
											FB_In.Teach_Servo_HomePos[Axis_Index] AND
											FB_In.Home_Position_Switch[Axis_Index] AND NOT
											FB_In.Quick_Home_REQ[Axis_Index];
			SET_HomeTMR[Axis_Index]();

			(*User Specified, Non-Delayed Homing Routine*)
			RPulse[0].CLK:= FB_In.Enable_Motion[Axis_Index] AND
							FB_In.Quick_Home_REQ[Axis_Index] AND NOT
							FB_In.Teach_Servo_HomePos[Axis_Index] AND NOT
							SET_HomeTMR[Axis_Index].Q AND NOT
							Homed[Axis_Index];
			RPulse[0]();

			IF SET_HomeTMR[Axis_Index].Q
				THEN
					fb_Set_Home[Axis_Index].HomingMode:= MC_Direct;
					fb_Set_Home[Axis_Index].Position:=0.0;
					fb_Set_Home[Axis_Index].Execute:= TRUE;
			ELSIF RPulse[0].Q OR (fb_Set_Home[Axis_Index].Busy AND NOT FB_In.Teach_Servo_HomePos[Axis_Index] AND NOT fb_Set_Home[Axis_Index].Done)
				THEN
					fb_Set_Home[Axis_Index].HomingMode:= FB_In.Homing_Type[Axis_Index];
					fb_Set_Home[Axis_Index].bCalibrationCam:= FB_In.Home_Position_Switch[Axis_Index];
					fb_Set_Home[Axis_Index].Position:= FB_In.Homing_Offset[Axis_index];
					fb_Set_Home[Axis_Index].Execute:= TRUE;
			ELSE
					fb_Set_Home[Axis_Index].Execute:= FALSE;
			END_IF;

			IF (NOT FB_In.Axis_Is_Absolute[Axis_Index] AND fb_Set_Home[Axis_Index].Done AND NOT fb_Set_Home[Axis_Index].Error)
				THEN
					Homed[Axis_Index]:= TRUE;
			END_IF;

ELSE
	fb_Move_ABS[Axis_Index].Execute:= FALSE;
	fb_Move_VEL[Axis_Index].Execute:= FALSE;
	Step_Complete[Axis_Index]:= FALSE;
	Step_Running[Axis_Index]:= FALSE;

END_IF; (*End of AUTO Home Routine*)

		IF FB_In.Axis_Is_Absolute[Axis_Index]
			THEN
			Homed[Axis_Index]:= TRUE;
		END_IF;


IF Step_Complete[Axis_Index] AND Step_Running[Axis_Index] AND NOT FB_In.Start_Explicit_StepCall[Axis_Index]
	THEN
			Step_Complete[Axis_Index]:= FALSE;
			Step_Running[Axis_Index]:= FALSE;
END_IF;

IF NOT FB_In.Start_PlayBack[Axis_Index]
	THEN
		Cycle_Complete[Axis_Index]:=FALSE;
END_IF;

IF ((Current_Step_Pointer[Axis_Index] <1) OR (Current_Step_Pointer[Axis_Index] >15)) AND Homed[Axis_Index]
	THEN
		Current_Step_Pointer[Axis_Index]:= 1;
END_IF;



(*!!!!!!!!!!!!!!!!!!!!!!!!!!!!!!!!!!!!!!!!!!!!!!!!!!!!!!!!!!!!!!!!!!!!!!!!!!!!!!!!!!!!!!!!!!!!!!!!!!!!!!!!!!!!!!!!!!!!! Diags and Error Resets !!!!!!!!!!!!!!!!!!!!!!!!!!!!!!!!!!!!!!!!!!!!!!!!!!!!!!!!!!!!!!!!!!!!!!!!!!!!!!!!!!!!!!!!!!!!!!!!!!!!!!!!!*)
	IF FB_In.Option_Type=0
		THEN
		ResetReq[Axis_Index]:=FB_In.Error_Reset[Axis_Index];
		DiagReq[Axis_Index]:= In_Error[Axis_Index];
		AX5000_DiagReset();	(*Call Action*)

	ELSIF FB_In.Option_Type=10
		THEN
		(*Drive Error Reset*)
		FB_Reset[Axis_Index].Execute:= FB_In.Error_Reset[Axis_Index];
		FB_Reset[Axis_Index](Axis:= Axis[Axis_Index]);
		(*Drive Low Level Reset*)
		FB_SoE_Reset[Axis_Index].Execute:= FB_In.Error_Reset[Axis_Index];
		FB_SoE_Reset[Axis_Index](Axis:= Axis[Axis_Index]);
	END_IF;

(*$$$$$$$$$$$$$$$$$$$$$$$$$$$$$$$$$$$$$$$$$$$$$$ Transfer Standard Outputs $$$$$$$$$$$$$$$$$$$$$$$$$$$$$$$$$$$$$$$$$$$*)
	(*Send Current Mode*)
	In_Play_ACK[Axis_Index]:= In_Play[Axis_Index];
	In_Teach_ACK[Axis_Index]:= In_Teach[Axis_Index];
	(*Send Maximum Torque values to PDO variables*)
	Drive_BipolarTorque[Axis_Index]:= FB_In.Max_Torque[Axis_Index];


	(*Send Out Status Bit for Drive Ready*)
		ReadyFor_Motion[Axis_Index]:= FB_In.Enable_Motion[Axis_Index] AND fb_Power[Axis_Index].Active AND NOT In_Error[Axis_Index] AND Homed[Axis_Index] AND
									fb_Power[Axis_Index].Status AND In_StandStill[Axis_Index] AND NOT fb_Stop[Axis_Index].Execute AND NOT fb_Stop[Axis_Index].Busy;
		ReadyFor_TeachMotion[Axis_Index]:= FB_In.Enable_Motion[Axis_Index] AND fb_Power[Axis_Index].Active AND NOT In_Error[Axis_Index]
											AND fb_Power[Axis_Index].Status AND NOT fb_Stop[Axis_Index].Execute AND NOT fb_Stop[Axis_Index].Busy;

	(*Send Drive_Read Information*)
		IF fb_Read_Status[Axis_Index].Valid
			THEN
				In_Error[Axis_Index]:= fb_Read_Status[Axis_Index].Error OR fb_Read_Status[Axis_Index].Status.Error;
				Error_ID[Axis_Index]:= fb_Read_Status[Axis_Index].ErrorID;
				In_Motion[Axis_Index]:= fb_Read_Status[Axis_Index].Status.Moving;
				In_Requested_Position[Axis_Index]:= (fb_Read_Status[Axis_Index].Status.InTargetPosition OR fb_Read_Status[Axis_Index].Status.InPositionArea)
											AND ((Current_Position[Axis_Index]+0.4)>= Program_Positions[Axis_Index][Current_Step_Pointer[Axis_Index]].Position)
											AND ((Current_Position[Axis_Index]-0.4)<= Program_Positions[Axis_Index][Current_Step_Pointer[Axis_Index]].Position);
				In_StandStill[Axis_Index]:= fb_Read_Status[Axis_Index].StandStill;
				In_Stopping[Axis_Index]:= fb_Read_Status[Axis_Index].Stopping;


		ELSE
				In_Motion[Axis_Index]:= FALSE;
				In_Requested_Position[Axis_Index]:= FALSE;

		END_IF;


	 (*Send Confirmation of At Requested Step*)
		IF In_Requested_Position[Axis_Index] AND NOT In_Motion[Axis_Index]
			THEN
			At_Current_Step[Axis_Index]:= Current_Step_Pointer[Axis_Index];
		ELSE
			At_Current_Step[Axis_Index]:= 0;
		END_IF;


	(*Send Positional Information*)
		IF Program_Positions[Axis_Index][Current_Step_Pointer[Axis_Index]].Move_Type<>3
			THEN
			Current_Position[Axis_Index]:= fb_Actual_Position[Axis_Index].Position;
		ELSIF (Program_Positions[Axis_Index][Current_Step_Pointer[Axis_Index]].Move_Type=3) OR Fb_In.Axis_Is_Absolute[Axis_Index]
			THEN
			Current_Position[Axis_Index]:= Axis[Axis_Index].NcToPlc.ModuloActPos;
		END_IF;

	(*Package Data to Move up to UI*)
		(*Type selection dependant data tranfer*)
		IF FB_In.Option_Type = 0	(*Default AX5206 type selected*)
			THEN
			Discrete_Image.AX5xxx:= Drive;
			Discrete_Image.AX5805:= Drive_AX5805;
			Discrete_Image.Safety_DIAG:= fb_AX5805_Info.Data;
			(*Drive and Motor Information*)
			Discrete_Image.Drive_Type_Message[Axis_Index]:= ST_Ax5000_Diag[Axis_Index].strDriveType;
			Discrete_Image.Axis_Motor_Message[Axis_Index]:= ST_AX5000_Diag[Axis_Index].strMotorType;
			(*Drive Level Operational State*)
			Discrete_Image.Drive_OperationalState[Axis_Index]:= ST_AX5000_Diag[Axis_Index].stDriveStatus.eActOpMode;
			(*Drive Level Errors*)
			Discrete_Image.Drive_In_Error[Axis_Index]:= NOT ST_AX5000_Diag[Axis_Index].stDriveStatus.bReadyForEnable OR
													ST_AX5000_Diag[Axis_Index].bC1DError OR NOT Homed[Axis_Index];

			Discrete_Image.Drive_Status[Axis_Index]:= ST_Ax5000_Diag[Axis_Index].wDriveStatus;
			Discrete_Image.Drive_StatusStruct[Axis_Index]:= ST_Ax5000_Diag[Axis_Index].stDriveStatus;
			Discrete_Image.Drive_Status_Message[Axis_Index]:= 'Test Drive Status Message';
			Discrete_Image.Drive_Diag_ErrorID[Axis_Index]:= ST_Ax5000_Diag[Axis_Index].iDiagNumber;
			Discrete_Image.Drive_Diag_Message[Axis_Index]:= ST_Ax5000_Diag[Axis_Index].strDiagMessageFull;
			Discrete_Image.Drive_C1D_ErrorID[Axis_Index]:= ST_Ax5000_Diag[Axis_Index].wClass1Diag;
			Discrete_Image.Drive_C1D_ErrorStruct[Axis_Index]:= ST_Ax5000_Diag[Axis_Index].stClass1Diag;
			Discrete_Image.Drive_C1D_Error_Message[Axis_Index]:= 'Test C1D Message';
			Discrete_Image.Axis_In_Error[Axis_Index]:= In_Error[Axis_Index];
			Discrete_Image.Axis_ErrorID[Axis_Index]:= Error_ID[Axis_Index];
			Discrete_Image.Axis_ErrorMessage[Axis_Index]:= FUN_GTAC_NC_Error_Messages(Error_ID[Axis_Index]);

		ELSIF FB_In.Option_Type = 10 (*EL7211 type selected*)
			THEN
			Discrete_Image.EL7xxx:=T03;
			(*NOTE, more error messaging and ID passing will have to be added with further testing of terminal drive, b.lekx-toniolo*)
		END_IF;
		(*Type independant data*)
		Discrete_Image.In_Play_ACK[Axis_Index]:= In_Play_ACK[Axis_Index];
		Discrete_Image.In_Teach_ACK[Axis_Index]:= In_Teach_ACK[Axis_Index];
		Discrete_Image.Current_Step_Pointer[Axis_Index]:= Current_Step_Pointer[Axis_Index];
		Discrete_Image.At_Current_Step[Axis_Index]:= At_Current_Step[Axis_Index];
		(*Tranfer Actual Step Data*)
		IF Current_Step_Pointer[Axis_Index]>1
			THEN
			Discrete_Image.Prev_Step_Data[Axis_Index]:= Program_Positions[Axis_Index][Current_Step_Pointer[Axis_Index]-1];
		ELSE
			Discrete_Image.Prev_Step_Data[Axis_Index]:= Program_Positions[Axis_Index][0];
		END_IF;
		Discrete_Image.Current_Step_Data[Axis_Index]:= Program_Positions[Axis_Index][Current_Step_Pointer[Axis_Index]];
		IF Current_Step_Pointer[Axis_Index]<15
			THEN
			Discrete_Image.Next_Step_Data[Axis_Index]:= Program_Positions[Axis_Index][Current_Step_Pointer[Axis_Index]+1];
		ELSE
			Discrete_Image.Next_Step_Data[Axis_Index]:= Program_Positions[Axis_Index][0];
		END_IF;

		Discrete_Image.Axis_Common_Name[Axis_Index]:= FB_In.Axis_Common_Name[Axis_Index];
		Discrete_Image.Corrected_Position[Axis_Index]:= Corrected_Position[Axis_Index];
		Discrete_Image.Actual_Position[Axis_Index]:= Current_Position[Axis_Index];
		Discrete_Image.In_Requested_Position[Axis_Index]:=In_Requested_Position[Axis_Index];
		Discrete_Image.In_Motion:= In_Motion;
		Discrete_Image.Is_Calibrated[Axis_Index]:= Homed[Axis_Index];
		Discrete_Image.Homed[Axis_Index]:= Homed[Axis_Index];
		Discrete_Image.Ready[Axis_Index]:=(In_Play_ACK[Axis_Index] AND ReadyFor_Motion[Axis_Index]) OR (In_Teach_ACK[Axis_Index] AND ReadyFor_TeachMotion[Axis_Index]) ;
		Discrete_Image.Software_Limit_Exceeded[Axis_Index]:= fb_Read_Status[Axis_Index].Status.SoftLimitMaxExceeded OR fb_Read_Status[Axis_Index].Status.SoftLimitMinExceeded;
		Discrete_Image.StateDWord[Axis_Index]:=Axis[Axis_Index].NcToPlc.StateDWord;
		Discrete_Image.Teach_Enable[Axis_Index]:=FB_In.Teach_Enable[Axis_Index];


END_FOR; (*End of Axis Index Loop*)

ACTION AX5000_DiagReset:
(* clear active flags for reset/diag *)
ResetAct[Axis_Index]:= FALSE;
DiagAct[Axis_Index]:= FALSE;

(* Diag + Reset of AX5000 *)
	(* call drive diag FBs *)
	fb_Axis_Diag[Axis_Index](
		IPCNetID	:= '',
		Axis		:= Axis[Axis_Index],
		stAX5000Diag:= ST_AX5000_Diag[Axis_Index],
		Reset   	:= ResetReq[Axis_Index],
		GetDiag 	:= DiagReq[Axis_Index]
	);

	(* update active flags for reset/diag *)
	ResetAct[Axis_Index]	:= ResetAct[Axis_Index] OR FB_Axis_Diag[Axis_Index].ResetAct;
	DiagAct[Axis_Index] := DiagAct[Axis_Index] OR FB_Axis_Diag[Axis_Index].DiagAct;

(*Reset of AX5805 (if applicable) after all other errors are reset*)
	IF FB_In.Option_Type<>10
		THEN
		CASE Axis_Index OF 
		1:
		Drive_Ax5805_Reset:= FB_In.Enable_Motion[1] AND NOT In_Error[1] AND Discrete_Image.AX5805.Axis1_Error_Ack;
		2:
		Drive_Ax5805_Reset:= FB_In.Enable_Motion[2] AND NOT In_Error[2] AND Discrete_Image.AX5805.Axis2_Error_Ack;

		END_CASE;

	END_IF;

(* clear reset/diag request if not active *)
ResetReq[Axis_Index]	:= ResetReq[Axis_Index] AND ResetAct[Axis_Index];
DiagReq[Axis_Index]		:= DiagReq[Axis_Index] AND DiagAct[Axis_Index];
END_ACTION

ACTION Move_Absolute:
(*General Set-Up Parameters/Function calls for Servo Drive*)

